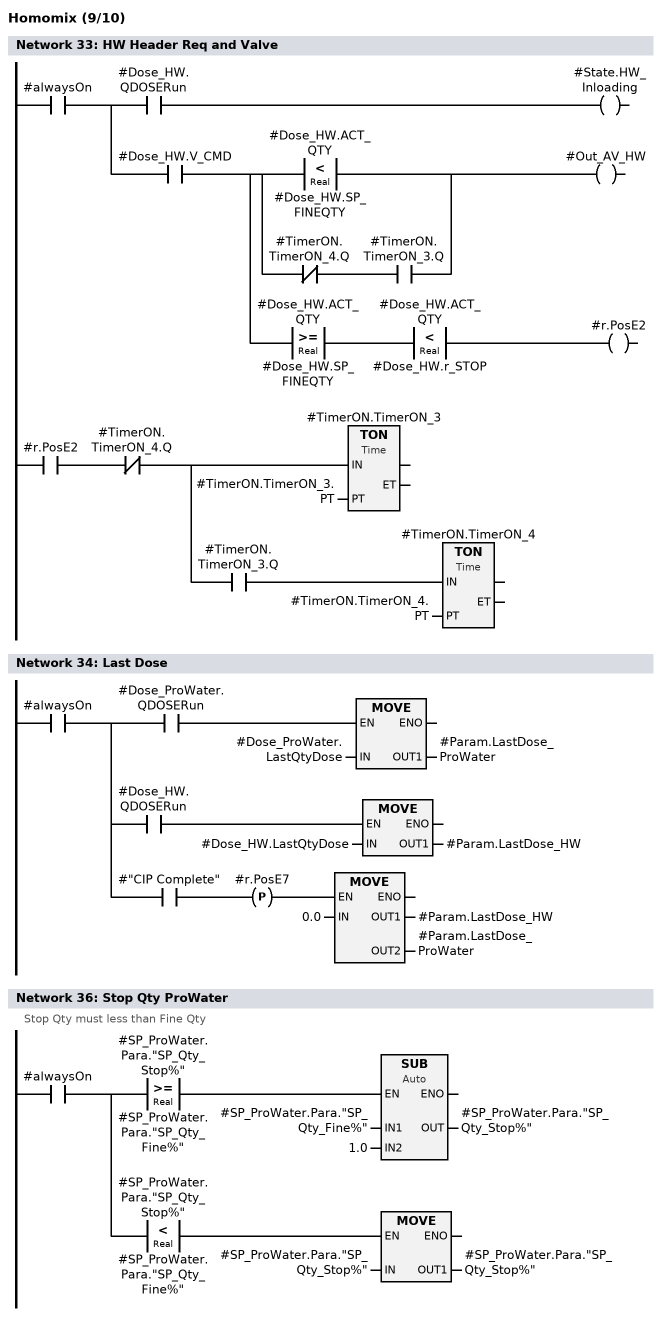
   RUNG wire#powerrail
      Contact( #alwaysOn )
      wire#w1
      Contact( #Dose_HW.QDOSERun )
      Coil( #State.HW_Inloading )
   END_RUNG
   RUNG wire#w1
      Contact( #Dose_HW.V_CMD )
      wire#w2
      { S7_Templates := "SrcType := Real" } LT_Contact(in1 := #Dose_HW.ACT_QTY, in2 := #Dose_HW.SP_FINEQTY)
      wire#w3
      Coil( #Out_AV_HW )
   END_RUNG
   RUNG wire#w2
      I_Contact( #TimerON.TimerON_4.Q )
      Contact( #TimerON.TimerON_3.Q )
   END_RUNG wire#w3
   RUNG wire#w2
      { S7_Templates := "SrcType := Real" } GE_Contact(in1 := #Dose_HW.ACT_QTY, in2 := #Dose_HW.SP_FINEQTY)
      { S7_Templates := "SrcType := Real" } LT_Contact(in1 := #Dose_HW.ACT_QTY, in2 := #Dose_HW.r_STOP)
      Coil( #r.PosE2 )
   END_RUNG
   RUNG wire#powerrail
      Contact( #r.PosE2 )
      I_Contact( #TimerON.TimerON_4.Q )
      wire#w4
      { S7_Templates := "time_type := Time" } #TimerON.TimerON_3.TON(pt := #TimerON.TimerON_3.PT, et =>)
   END_RUNG
   RUNG wire#w4
      Contact( #TimerON.TimerON_3.Q )
      { S7_Templates := "time_type := Time" } #TimerON.TimerON_4.TON(pt := #TimerON.TimerON_4.PT, et =>)
   END_RUNG
   // the same network as SCL:
   #State.HW_Inloading := #alwaysOn AND #Dose_HW.QDOSERun;
   #_w1 := #alwaysOn AND #Dose_HW.V_CMD;
   #Out_AV_HW := #_w1 AND ((#Dose_HW.ACT_QTY < #Dose_HW.SP_FINEQTY) OR (NOT #TimerON.TimerON_4.Q AND #TimerON.TimerON_3.Q));
   #r.PosE2 := #_w1 AND (#Dose_HW.ACT_QTY >= #Dose_HW.SP_FINEQTY) AND (#Dose_HW.ACT_QTY < #Dose_HW.r_STOP);
   #_w2 := #r.PosE2 AND NOT #TimerON.TimerON_4.Q;
   #TimerON.TimerON_3.TON(IN := #_w2, PT := #TimerON.TimerON_3.PT);
   #TimerON.TimerON_4.TON(IN := #_w2 AND #TimerON.TimerON_3.Q, PT := #TimerON.TimerON_4.PT);
END_REGION

REGION Network 34: Last Dose
   RUNG wire#powerrail
      Contact( #alwaysOn )
      wire#w1
      Contact( #Dose_ProWater.QDOSERun )
      Move(in := #Dose_ProWater.LastQtyDose, out1 => #Param.LastDose_ProWater)
   END_RUNG
   RUNG wire#w1
      Contact( #Dose_HW.QDOSERun )
      Move(in := #Dose_HW.LastQtyDose, out1 => #Param.LastDose_HW)
   END_RUNG
   RUNG wire#w1
      Contact( #"CIP Complete" )
      P_Trig( #r.PosE7 )
      Move(in := 0.0, out1 => #Param.LastDose_HW, out2 => #Param.LastDose_ProWater)
   END_RUNG
   // the same network as SCL:
   IF #alwaysOn AND #Dose_ProWater.QDOSERun THEN
       #Param.LastDose_ProWater := #Dose_ProWater.LastQtyDose;
   END_IF;
   IF #alwaysOn AND #Dose_HW.QDOSERun THEN #Param.LastDose_HW := #Dose_HW.LastQtyDose; END_IF;
   #_w1 := #alwaysOn AND #"CIP Complete";
   #_w2 := #_w1 AND NOT #r.PosE7;   // rising edge
   #r.PosE7 := #_w1;
   IF #_w2 THEN
       #Param.LastDose_HW := 0.0;
       #Param.LastDose_ProWater := 0.0;
   END_IF;
END_REGION

REGION Network 36: Stop Qty ProWater
   // Stop Qty must less than Fine Qty
   RUNG wire#powerrail
      Contact( #alwaysOn )
      wire#w1
      { S7_Templates := "SrcType := Real" } GE_Contact(in1 := #SP_ProWater.Para."SP_Qty_Stop%", in2 := #SP_ProWater.Para."SP_Qty_Fine%")
      Sub(in1 := #SP_ProWater.Para."SP_Qty_Fine%", in2 := 1.0, out => #SP_ProWater.Para."SP_Qty_Stop%")
   END_RUNG
   RUNG wire#w1
      { S7_Templates := "SrcType := Real" } LT_Contact(in1 := #SP_ProWater.Para."SP_Qty_Stop%", in2 := #SP_ProWater.Para."SP_Qty_Fine%")
      Move(in := #SP_ProWater.Para."SP_Qty_Stop%", out1 => #SP_ProWater.Para."SP_Qty_Stop%")
   END_RUNG
   // the same network as SCL:
   IF #alwaysOn AND (#SP_ProWater.Para."SP_Qty_Stop%" >= #SP_ProWater.Para."SP_Qty_Fine%") THEN
       #SP_ProWater.Para."SP_Qty_Stop%" := #SP_ProWater.Para."SP_Qty_Fine%" - 1.0;
   END_IF;
   IF #alwaysOn AND (#SP_ProWater.Para."SP_Qty_Stop%" < #SP_ProWater.Para."SP_Qty_Fine%") THEN
       #SP_ProWater.Para."SP_Qty_Stop%" := #SP_ProWater.Para."SP_Qty_Stop%";
   END_IF;
END_REGION

REGION Network 37: Stop Qty HW
   // Stop Qty must less than Fine Qty
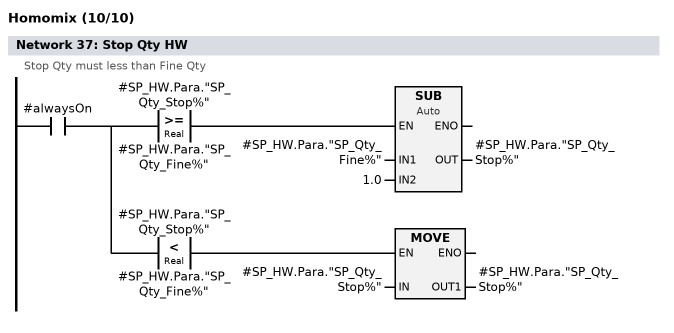
   RUNG wire#powerrail
      Contact( #alwaysOn )
      wire#w1
      { S7_Templates := "SrcType := Real" } GE_Contact(in1 := #SP_HW.Para."SP_Qty_Stop%", in2 := #SP_HW.Para."SP_Qty_Fine%")
      Sub(in1 := #SP_HW.Para."SP_Qty_Fine%", in2 := 1.0, out => #SP_HW.Para."SP_Qty_Stop%")
   END_RUNG
   RUNG wire#w1
      { S7_Templates := "SrcType := Real" } LT_Contact(in1 := #SP_HW.Para."SP_Qty_Stop%", in2 := #SP_HW.Para."SP_Qty_Fine%")
      Move(in := #SP_HW.Para."SP_Qty_Stop%", out1 => #SP_HW.Para."SP_Qty_Stop%")
   END_RUNG
   // the same network as SCL:
   IF #alwaysOn AND (#SP_HW.Para."SP_Qty_Stop%" >= #SP_HW.Para."SP_Qty_Fine%") THEN
       #SP_HW.Para."SP_Qty_Stop%" := #SP_HW.Para."SP_Qty_Fine%" - 1.0;
   END_IF;
   IF #alwaysOn AND (#SP_HW.Para."SP_Qty_Stop%" < #SP_HW.Para."SP_Qty_Fine%") THEN
       #SP_HW.Para."SP_Qty_Stop%" := #SP_HW.Para."SP_Qty_Stop%";
   END_IF;
END_REGION
END_FUNCTION_BLOCK

FUNCTION_BLOCK "Raw_Pulse"   // FB20, LAD
{ S7_Optimized_Access := 'TRUE' }
VERSION : 0.1
// stored: AutoNumber true, IsIECCheckEnabled false, IsRetainMemResEnabled false, MemoryReserve 100, SetENOAutomatically false, UDAEnableTagReadback false
   VAR_INPUT
      CountReset : Bool;
      CountMode : Bool;
      DoseRun : Bool;
      CmdStep : Int;
      FT_Pulse : Bool;   // Pulse Flow Meter
      FT_Tot : Real;
      Dose_SP : Real;
      Speed_AV : Real;
      Speed_SP : Real;
   END_VAR
   VAR_OUTPUT
      Q_FT_Star : Real;
      Q_FT_Stop : Real;
      Q_SPQty : Real;
      Q_FineQty : Real;
      Q_StopQty : Real;
      Q_P_Speed : Real;
      Q_P_FineSpeed : Real;
      Q_P_CoasSpeed : Real;
   END_VAR
   VAR_IN_OUT
      Q_FT_Tot : Real;
   END_VAR
   VAR RETAIN
      Para : Struct
         "SP_Qty_Stop%" : Real := 3.0;
         "SP_Qty_Fine%" : Real := 20.0;
         SP_Qty_Stop : Real;
         SP_Qty_Fine : Real;
         SP_Pump_Co : Real := 80.0;
         SP_Pump_Fi : Real := 20.0;
         "Pulse/Liter" : Real := 1.0;
      END_STRUCT;
   END_VAR
   VAR
      alwaysON { S7_SetPoint := 'True'} : Bool;
      DosePE : Bool;
      "BIT.FT_Pulse" : Bool;
   END_VAR
   VAR_TEMP   // added for the SCL form of the ladder/FBD networks
      _w1 : Bool;
      _w2 : Bool;
      _w3 : Bool;
      _w4 : Bool;
   END_VAR
BEGIN

REGION Network 1: alwaysON
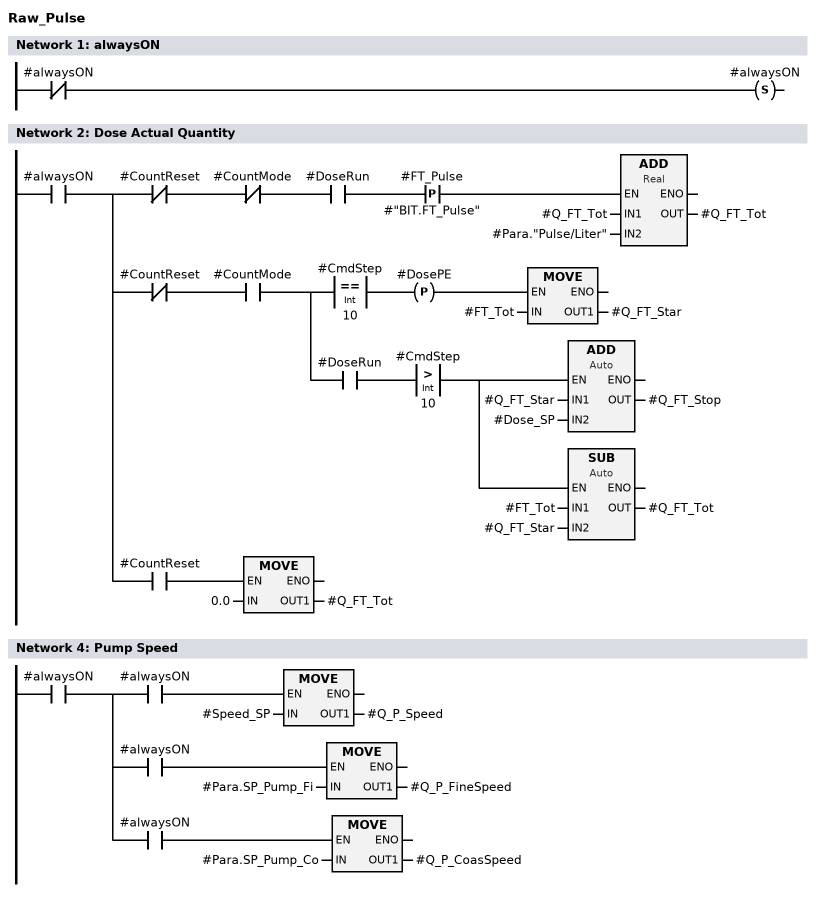
   RUNG wire#powerrail
      I_Contact( #alwaysON )
      S_Coil( #alwaysON )
   END_RUNG
   // the same network as SCL:
   IF NOT #alwaysON THEN #alwaysON := TRUE; END_IF;
END_REGION

REGION Network 2: Dose Actual Quantity
   RUNG wire#powerrail
      Contact( #alwaysON )
      wire#w1
      I_Contact( #CountReset )
      I_Contact( #CountMode )
      Contact( #DoseRun )
      P_Contact(operand := #FT_Pulse, bit := #"BIT.FT_Pulse")
      { S7_Templates := "SrcType := Real" } Add(in1 := #Q_FT_Tot, in2 := #Para."Pulse/Liter", out => #Q_FT_Tot)
   END_RUNG
   RUNG wire#w1
      I_Contact( #CountReset )
      Contact( #CountMode )
      wire#w2
      { S7_Templates := "SrcType := Int" } EQ_Contact(in1 := #CmdStep, in2 := 10)
      P_Trig( #DosePE )
      Move(in := #FT_Tot, out1 => #Q_FT_Star)
   END_RUNG
   RUNG wire#w2
      Contact( #DoseRun )
      { S7_Templates := "SrcType := Int" } GT_Contact(in1 := #CmdStep, in2 := 10)
      wire#w3
      Add(in1 := #Q_FT_Star, in2 := #Dose_SP, out => #Q_FT_Stop)
   END_RUNG
   RUNG wire#w3
      Sub(in1 := #FT_Tot, in2 := #Q_FT_Star, out => #Q_FT_Tot)
   END_RUNG
   RUNG wire#w1
      Contact( #CountReset )
      Move(in := 0.0, out1 => #Q_FT_Tot)
   END_RUNG
   // the same network as SCL:
   #_w1 := #alwaysON AND NOT #CountReset AND NOT #CountMode AND #DoseRun AND #FT_Pulse AND NOT #"BIT.FT_Pulse";   // rising edge of #FT_Pulse
   #"BIT.FT_Pulse" := #FT_Pulse;
   IF #_w1 THEN #Q_FT_Tot := #Q_FT_Tot + #Para."Pulse/Liter"; END_IF;
   #_w2 := #alwaysON AND NOT #CountReset AND #CountMode;
   #_w3 := #_w2 AND (#CmdStep = 10);
   #_w4 := #_w3 AND NOT #DosePE;   // rising edge
   #DosePE := #_w3;
   IF #_w4 THEN #Q_FT_Star := #FT_Tot; END_IF;
   IF #_w2 AND #DoseRun AND (#CmdStep > 10) THEN
       #Q_FT_Stop := #Q_FT_Star + #Dose_SP;
       #Q_FT_Tot := #FT_Tot - #Q_FT_Star;
   END_IF;
   IF #alwaysON AND #CountReset THEN #Q_FT_Tot := 0.0; END_IF;
END_REGION

NETWORK
TITLE = Quantity Calculation
// SP Quantity
      L     #Dose_SP;
      T     #Q_SPQty;
// Fine Quantity Calculation
      L     #Dose_SP;
      L     #Para."SP_Qty_Fine%";
      *R;
      L     100.0;
      /R;
      T     #Para.SP_Qty_Fine;

      L     #Dose_SP;
      L     #Para.SP_Qty_Fine;
      -R;
      T     #Q_FineQty;

// Stop Quantity Calculation
      L     #Dose_SP;
      L     #Para."SP_Qty_Stop%";
      *R;
      L     100.0;
      /R;
      T     #Para.SP_Qty_Stop;

      L     #Dose_SP;
      L     #Para.SP_Qty_Stop;
      -R;
      T     #Q_StopQty;


REGION Network 4: Pump Speed
   RUNG wire#powerrail
      Contact( #alwaysON )
      wire#w1
      Contact( #alwaysON )
      Move(in := #Speed_SP, out1 => #Q_P_Speed)
   END_RUNG
   RUNG wire#w1
      Contact( #alwaysON )
      Move(in := #Para.SP_Pump_Fi, out1 => #Q_P_FineSpeed)
   END_RUNG
   RUNG wire#w1
      Contact( #alwaysON )
      Move(in := #Para.SP_Pump_Co, out1 => #Q_P_CoasSpeed)
   END_RUNG
   // the same network as SCL:
   IF #alwaysON AND #alwaysON THEN
       #Q_P_Speed := #Speed_SP;
       #Q_P_FineSpeed := #Para.SP_Pump_Fi;
       #Q_P_CoasSpeed := #Para.SP_Pump_Co;
   END_IF;
END_REGION
END_FUNCTION_BLOCK

FUNCTION_BLOCK "IO Valve Homomixer"   // FB3, LAD
{ S7_Optimized_Access := 'FALSE' }
VERSION : 0.1
// stored: AutoNumber true, IsIECCheckEnabled false, SetENOAutomatically false, UDAEnableTagReadback false
   VAR_INPUT
      lock : Bool;
      Init : Bool;
      testing : Bool;
      Reset : Bool;
   END_VAR
   VAR
      "AV-12.01" { S7_SetPoint := 'True'} : "Valve";
      "AV-12.02" { S7_SetPoint := 'True'} : "Valve";
      "AV-12.03" { S7_SetPoint := 'True'} : "Valve";
      "AV-12.04" { S7_SetPoint := 'True'} : "Valve";
      "AV-12.05" { S7_SetPoint := 'True'} : "Valve";
      "AV-12.06" { S7_SetPoint := 'True'} : "Valve";
      "AV-12.07" { S7_SetPoint := 'True'} : "Valve";
      "AV-12.11" { S7_SetPoint := 'True'} : "Valve";
      "AV-12.12" { S7_SetPoint := 'True'} : "Valve";
      "AV-13.01" { S7_SetPoint := 'True'} : "Valve";
      "AV-13.02" { S7_SetPoint := 'True'} : "Valve";
      "AV-13.03" { S7_SetPoint := 'True'} : "Valve";
      "AV-13.04" { S7_SetPoint := 'True'} : "Valve";
      "AV-13.05" { S7_SetPoint := 'True'} : "Valve";
      "AV-13.06" { S7_SetPoint := 'True'} : "Valve";
      "AV-13.07" { S7_SetPoint := 'True'} : "Valve";
      "AV-14.01" { S7_SetPoint := 'True'} : "Valve";
      "AV-14.02" { S7_SetPoint := 'True'} : "Valve";
      "AV-14.03" { S7_SetPoint := 'True'} : "Valve";
      "AV-14.04" { S7_SetPoint := 'True'} : "Valve";
      "AV-14.05" { S7_SetPoint := 'True'} : "Valve";
      "AV-14.06" { S7_SetPoint := 'True'} : "Valve";
      "AV-14.07" { S7_SetPoint := 'True'} : "Valve";
      "P-12.01" { S7_SetPoint := 'True'} : "Motor";
      "P-13.01" { S7_SetPoint := 'True'} : "Motor";
      "P-14.01" { S7_SetPoint := 'True'} : "Motor";
   END_VAR
   // "AV-12.01".OPdwCmd := 16#0008_0000;
   // "AV-12.02".OPdwCmd := 16#0008_0000;
   // "AV-12.03".OPdwCmd := 16#0002_0000;
   // "AV-12.04".OPdwCmd := 16#0008_0000;
   // "AV-13.01".OPdwCmd := 16#0008_0000;
   // "AV-13.02".OPdwCmd := 16#0008_0000;
   // "AV-13.03".OPdwCmd := 16#0002_0000;
BEGIN

REGION Network 1 (SCL): FB OPEN and CLOSE 12
   IF #testing THEN
       // Statement section IF
       #"AV-12.01".FB_OPEN := #"AV-12.01".QCMD_OP;
       #"AV-12.01".FB_CLOSE := NOT #"AV-12.01".QCMD_OP;
       #"AV-12.02".FB_OPEN := #"AV-12.02".QCMD_OP;
       #"AV-12.02".FB_CLOSE := NOT #"AV-12.02".QCMD_OP;
       #"AV-12.03".FB_OPEN := #"AV-12.03".QCMD_OP;
       #"AV-12.03".FB_CLOSE := NOT #"AV-12.03".QCMD_OP;
       #"AV-12.04".FB_OPEN := #"AV-12.04".QCMD_OP;
       #"AV-12.04".FB_CLOSE := NOT #"AV-12.04".QCMD_OP;
       #"AV-12.05".FB_OPEN := #"AV-12.05".QCMD_OP;
       #"AV-12.05".FB_CLOSE := NOT #"AV-12.05".QCMD_OP;
       #"AV-12.06".FB_OPEN := #"AV-12.06".QCMD_OP;
       #"AV-12.06".FB_CLOSE := NOT #"AV-12.06".QCMD_OP;
       #"AV-12.07".FB_OPEN := #"AV-12.07".QCMD_OP;
       #"AV-12.07".FB_CLOSE := NOT #"AV-12.07".QCMD_OP;
       #"AV-12.11".FB_OPEN := #"AV-12.11".QCMD_OP;
       #"AV-12.11".FB_CLOSE := NOT #"AV-12.11".QCMD_OP;
       #"AV-12.12".FB_OPEN := #"AV-12.12".QCMD_OP;
       #"AV-12.12".FB_CLOSE := NOT #"AV-12.12".QCMD_OP;
   ELSE
       // Statement section ELSE
       #"AV-12.01".FB_OPEN := NOT "ZSC-12.01";
       #"AV-12.01".FB_CLOSE := "ZSC-12.01";
       #"AV-12.02".FB_OPEN := NOT "ZSC-12.02";
       #"AV-12.02".FB_CLOSE := "ZSC-12.02";
       #"AV-12.03".FB_OPEN := #"AV-12.03".QCMD_OP;
       #"AV-12.03".FB_CLOSE := NOT #"AV-12.03".QCMD_OP;
       #"AV-12.04".FB_OPEN := #"AV-12.04".QCMD_OP;
       #"AV-12.04".FB_CLOSE := NOT #"AV-12.04".QCMD_OP;
       #"AV-12.05".FB_OPEN := #"AV-12.05".QCMD_OP;
       #"AV-12.05".FB_CLOSE := NOT #"AV-12.05".QCMD_OP;
       #"AV-12.06".FB_OPEN := #"AV-12.06".QCMD_OP;
       #"AV-12.06".FB_CLOSE := NOT #"AV-12.06".QCMD_OP;
       #"AV-12.07".FB_OPEN := #"AV-12.07".QCMD_OP;
       #"AV-12.07".FB_CLOSE := NOT #"AV-12.07".QCMD_OP;
       #"AV-12.11".FB_OPEN := #"AV-12.11".QCMD_OP;
       #"AV-12.11".FB_CLOSE := NOT #"AV-12.11".QCMD_OP;
       #"AV-12.12".FB_OPEN := #"AV-12.12".QCMD_OP;
       #"AV-12.12".FB_CLOSE := NOT #"AV-12.12".QCMD_OP;
   END_IF;
END_REGION

NETWORK
TITLE = FB Monitoring Time 12
// FB OPEN Time
      L     t#20s;
      T     #"AV-12.01".MON_T;
      T     #"AV-12.02".MON_T;
      T     #"AV-12.03".MON_T;
      T     #"AV-12.04".MON_T;
      T     #"AV-12.05".MON_T;
      T     #"AV-12.06".MON_T;
      T     #"AV-12.07".MON_T;
      T     #"AV-12.11".MON_T;
      T     #"AV-12.12".MON_T;
// FB CLOSE Time
      L     t#20s;
      T     #"AV-12.01".MON_T_CLOSE;
      T     #"AV-12.02".MON_T_CLOSE;
      T     #"AV-12.03".MON_T_CLOSE;
      T     #"AV-12.04".MON_T_CLOSE;
      T     #"AV-12.05".MON_T_CLOSE;
      T     #"AV-12.06".MON_T_CLOSE;
      T     #"AV-12.07".MON_T_CLOSE;
      T     #"AV-12.11".MON_T_CLOSE;
      T     #"AV-12.12".MON_T_CLOSE;

REGION Network 3: AV-12.01 w ZSC
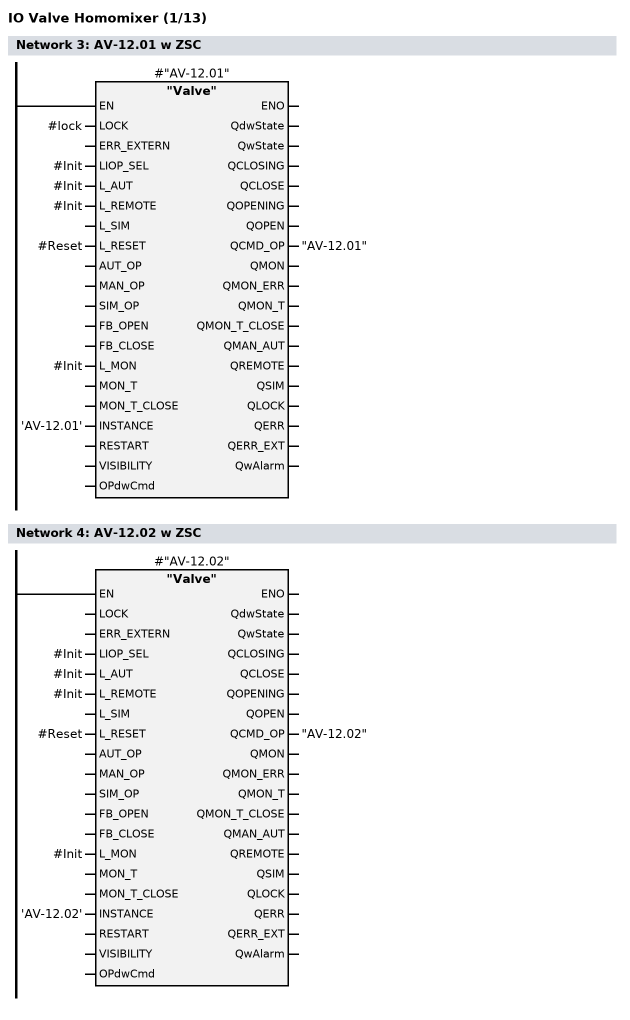
   RUNG wire#powerrail
      #"AV-12.01"(LOCK := #lock, ERR_EXTERN :=, LIOP_SEL := #Init, L_AUT := #Init, L_REMOTE := #Init, L_SIM :=, L_RESET := #Reset, AUT_OP :=, MAN_OP :=, SIM_OP :=, FB_OPEN :=, FB_CLOSE :=, L_MON := #Init, MON_T :=, MON_T_CLOSE :=, INSTANCE := 'AV-12.01', RESTART :=, VISIBILITY :=, OPdwCmd :=, QdwState =>, QwState =>, QCLOSING =>, QCLOSE =>, QOPENING =>, QOPEN =>, QCMD_OP => "AV-12.01", QMON =>, QMON_ERR =>, QMON_T =>, QMON_T_CLOSE =>, QMAN_AUT =>, QREMOTE =>, QSIM =>, QLOCK =>, QERR =>, QERR_EXT =>, QwAlarm =>)
   END_RUNG
   // the same network as SCL:
   #"AV-12.01"(LOCK := #lock,   // "Valve"
               LIOP_SEL := #Init,
               L_AUT := #Init,
               L_REMOTE := #Init,
               L_RESET := #Reset,
               L_MON := #Init,
               INSTANCE := 'AV-12.01',
               QCMD_OP => "AV-12.01");
END_REGION

REGION Network 4: AV-12.02 w ZSC
   RUNG wire#powerrail
      #"AV-12.02"(LOCK :=, ERR_EXTERN :=, LIOP_SEL := #Init, L_AUT := #Init, L_REMOTE := #Init, L_SIM :=, L_RESET := #Reset, AUT_OP :=, MAN_OP :=, SIM_OP :=, FB_OPEN :=, FB_CLOSE :=, L_MON := #Init, MON_T :=, MON_T_CLOSE :=, INSTANCE := 'AV-12.02', RESTART :=, VISIBILITY :=, OPdwCmd :=, QdwState =>, QwState =>, QCLOSING =>, QCLOSE =>, QOPENING =>, QOPEN =>, QCMD_OP => "AV-12.02", QMON =>, QMON_ERR =>, QMON_T =>, QMON_T_CLOSE =>, QMAN_AUT =>, QREMOTE =>, QSIM =>, QLOCK =>, QERR =>, QERR_EXT =>, QwAlarm =>)
   END_RUNG
   // the same network as SCL:
   #"AV-12.02"(LIOP_SEL := #Init,   // "Valve"
               L_AUT := #Init,
               L_REMOTE := #Init,
               L_RESET := #Reset,
               L_MON := #Init,
               INSTANCE := 'AV-12.02',
               QCMD_OP => "AV-12.02");
END_REGION

REGION Network 5: AV-12.03
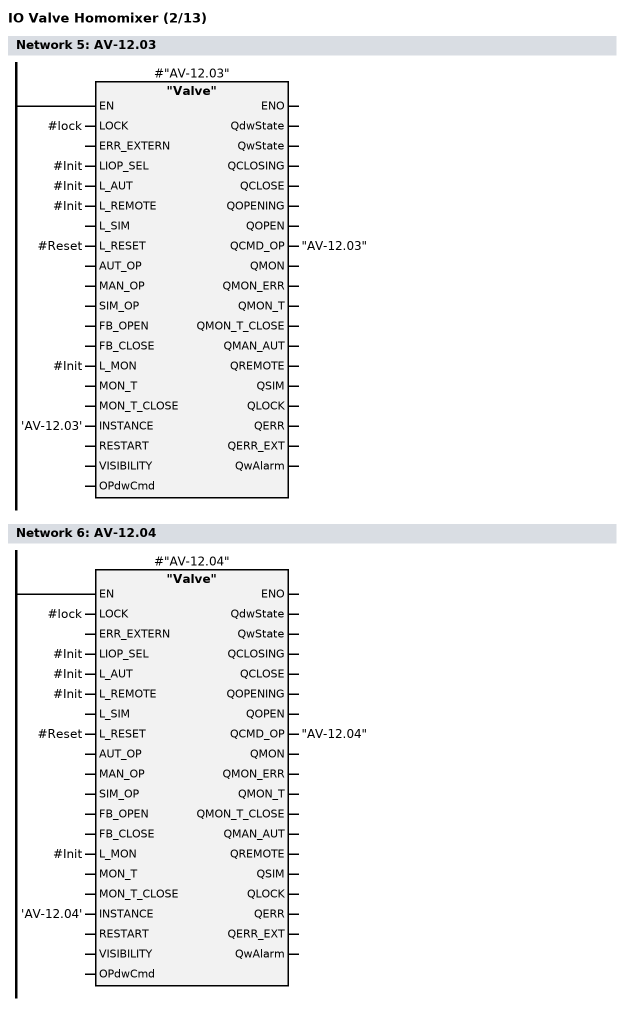
   RUNG wire#powerrail
      #"AV-12.03"(LOCK := #lock, ERR_EXTERN :=, LIOP_SEL := #Init, L_AUT := #Init, L_REMOTE := #Init, L_SIM :=, L_RESET := #Reset, AUT_OP :=, MAN_OP :=, SIM_OP :=, FB_OPEN :=, FB_CLOSE :=, L_MON := #Init, MON_T :=, MON_T_CLOSE :=, INSTANCE := 'AV-12.03', RESTART :=, VISIBILITY :=, OPdwCmd :=, QdwState =>, QwState =>, QCLOSING =>, QCLOSE =>, QOPENING =>, QOPEN =>, QCMD_OP => "AV-12.03", QMON =>, QMON_ERR =>, QMON_T =>, QMON_T_CLOSE =>, QMAN_AUT =>, QREMOTE =>, QSIM =>, QLOCK =>, QERR =>, QERR_EXT =>, QwAlarm =>)
   END_RUNG
   // the same network as SCL:
   #"AV-12.03"(LOCK := #lock,   // "Valve"
               LIOP_SEL := #Init,
               L_AUT := #Init,
               L_REMOTE := #Init,
               L_RESET := #Reset,
               L_MON := #Init,
               INSTANCE := 'AV-12.03',
               QCMD_OP => "AV-12.03");
END_REGION

REGION Network 6: AV-12.04
   RUNG wire#powerrail
      #"AV-12.04"(LOCK := #lock, ERR_EXTERN :=, LIOP_SEL := #Init, L_AUT := #Init, L_REMOTE := #Init, L_SIM :=, L_RESET := #Reset, AUT_OP :=, MAN_OP :=, SIM_OP :=, FB_OPEN :=, FB_CLOSE :=, L_MON := #Init, MON_T :=, MON_T_CLOSE :=, INSTANCE := 'AV-12.04', RESTART :=, VISIBILITY :=, OPdwCmd :=, QdwState =>, QwState =>, QCLOSING =>, QCLOSE =>, QOPENING =>, QOPEN =>, QCMD_OP => "AV-12.04", QMON =>, QMON_ERR =>, QMON_T =>, QMON_T_CLOSE =>, QMAN_AUT =>, QREMOTE =>, QSIM =>, QLOCK =>, QERR =>, QERR_EXT =>, QwAlarm =>)
   END_RUNG
   // the same network as SCL:
   #"AV-12.04"(LOCK := #lock,   // "Valve"
               LIOP_SEL := #Init,
               L_AUT := #Init,
               L_REMOTE := #Init,
               L_RESET := #Reset,
               L_MON := #Init,
               INSTANCE := 'AV-12.04',
               QCMD_OP => "AV-12.04");
END_REGION

REGION Network 7: AV-12.05
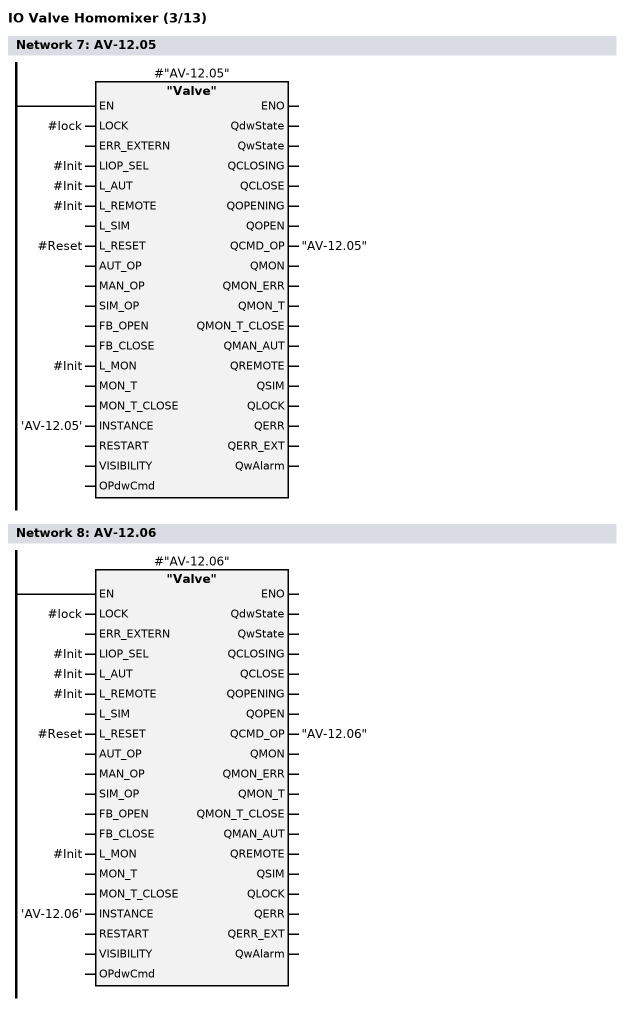
   RUNG wire#powerrail
      #"AV-12.05"(LOCK := #lock, ERR_EXTERN :=, LIOP_SEL := #Init, L_AUT := #Init, L_REMOTE := #Init, L_SIM :=, L_RESET := #Reset, AUT_OP :=, MAN_OP :=, SIM_OP :=, FB_OPEN :=, FB_CLOSE :=, L_MON := #Init, MON_T :=, MON_T_CLOSE :=, INSTANCE := 'AV-12.05', RESTART :=, VISIBILITY :=, OPdwCmd :=, QdwState =>, QwState =>, QCLOSING =>, QCLOSE =>, QOPENING =>, QOPEN =>, QCMD_OP => "AV-12.05", QMON =>, QMON_ERR =>, QMON_T =>, QMON_T_CLOSE =>, QMAN_AUT =>, QREMOTE =>, QSIM =>, QLOCK =>, QERR =>, QERR_EXT =>, QwAlarm =>)
   END_RUNG
   // the same network as SCL:
   #"AV-12.05"(LOCK := #lock,   // "Valve"
               LIOP_SEL := #Init,
               L_AUT := #Init,
               L_REMOTE := #Init,
               L_RESET := #Reset,
               L_MON := #Init,
               INSTANCE := 'AV-12.05',
               QCMD_OP => "AV-12.05");
END_REGION

REGION Network 8: AV-12.06
   RUNG wire#powerrail
      #"AV-12.06"(LOCK := #lock, ERR_EXTERN :=, LIOP_SEL := #Init, L_AUT := #Init, L_REMOTE := #Init, L_SIM :=, L_RESET := #Reset, AUT_OP :=, MAN_OP :=, SIM_OP :=, FB_OPEN :=, FB_CLOSE :=, L_MON := #Init, MON_T :=, MON_T_CLOSE :=, INSTANCE := 'AV-12.06', RESTART :=, VISIBILITY :=, OPdwCmd :=, QdwState =>, QwState =>, QCLOSING =>, QCLOSE =>, QOPENING =>, QOPEN =>, QCMD_OP => "AV-12.06", QMON =>, QMON_ERR =>, QMON_T =>, QMON_T_CLOSE =>, QMAN_AUT =>, QREMOTE =>, QSIM =>, QLOCK =>, QERR =>, QERR_EXT =>, QwAlarm =>)
   END_RUNG
   // the same network as SCL:
   #"AV-12.06"(LOCK := #lock,   // "Valve"
               LIOP_SEL := #Init,
               L_AUT := #Init,
               L_REMOTE := #Init,
               L_RESET := #Reset,
               L_MON := #Init,
               INSTANCE := 'AV-12.06',
               QCMD_OP => "AV-12.06");
END_REGION

REGION Network 9: AV-12.07
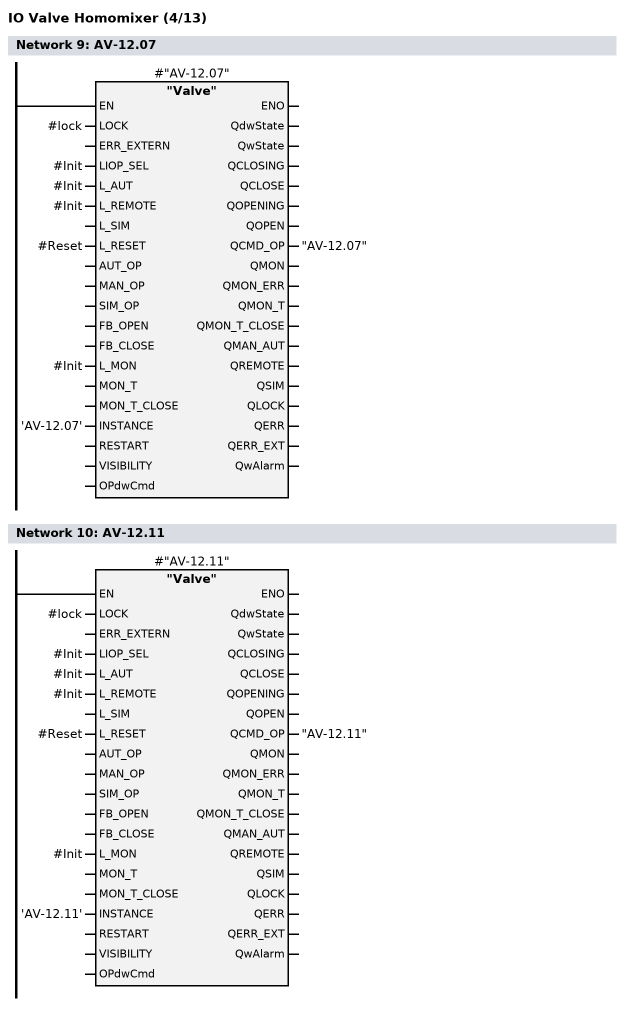
   RUNG wire#powerrail
      #"AV-12.07"(LOCK := #lock, ERR_EXTERN :=, LIOP_SEL := #Init, L_AUT := #Init, L_REMOTE := #Init, L_SIM :=, L_RESET := #Reset, AUT_OP :=, MAN_OP :=, SIM_OP :=, FB_OPEN :=, FB_CLOSE :=, L_MON := #Init, MON_T :=, MON_T_CLOSE :=, INSTANCE := 'AV-12.07', RESTART :=, VISIBILITY :=, OPdwCmd :=, QdwState =>, QwState =>, QCLOSING =>, QCLOSE =>, QOPENING =>, QOPEN =>, QCMD_OP => "AV-12.07", QMON =>, QMON_ERR =>, QMON_T =>, QMON_T_CLOSE =>, QMAN_AUT =>, QREMOTE =>, QSIM =>, QLOCK =>, QERR =>, QERR_EXT =>, QwAlarm =>)
   END_RUNG
   // the same network as SCL:
   #"AV-12.07"(LOCK := #lock,   // "Valve"
               LIOP_SEL := #Init,
               L_AUT := #Init,
               L_REMOTE := #Init,
               L_RESET := #Reset,
               L_MON := #Init,
               INSTANCE := 'AV-12.07',
               QCMD_OP => "AV-12.07");
END_REGION

REGION Network 10: AV-12.11
   RUNG wire#powerrail
      #"AV-12.11"(LOCK := #lock, ERR_EXTERN :=, LIOP_SEL := #Init, L_AUT := #Init, L_REMOTE := #Init, L_SIM :=, L_RESET := #Reset, AUT_OP :=, MAN_OP :=, SIM_OP :=, FB_OPEN :=, FB_CLOSE :=, L_MON := #Init, MON_T :=, MON_T_CLOSE :=, INSTANCE := 'AV-12.11', RESTART :=, VISIBILITY :=, OPdwCmd :=, QdwState =>, QwState =>, QCLOSING =>, QCLOSE =>, QOPENING =>, QOPEN =>, QCMD_OP => "AV-12.11", QMON =>, QMON_ERR =>, QMON_T =>, QMON_T_CLOSE =>, QMAN_AUT =>, QREMOTE =>, QSIM =>, QLOCK =>, QERR =>, QERR_EXT =>, QwAlarm =>)
   END_RUNG
   // the same network as SCL:
   #"AV-12.11"(LOCK := #lock,   // "Valve"
               LIOP_SEL := #Init,
               L_AUT := #Init,
               L_REMOTE := #Init,
               L_RESET := #Reset,
               L_MON := #Init,
               INSTANCE := 'AV-12.11',
               QCMD_OP => "AV-12.11");
END_REGION

REGION Network 11: AV-12.12
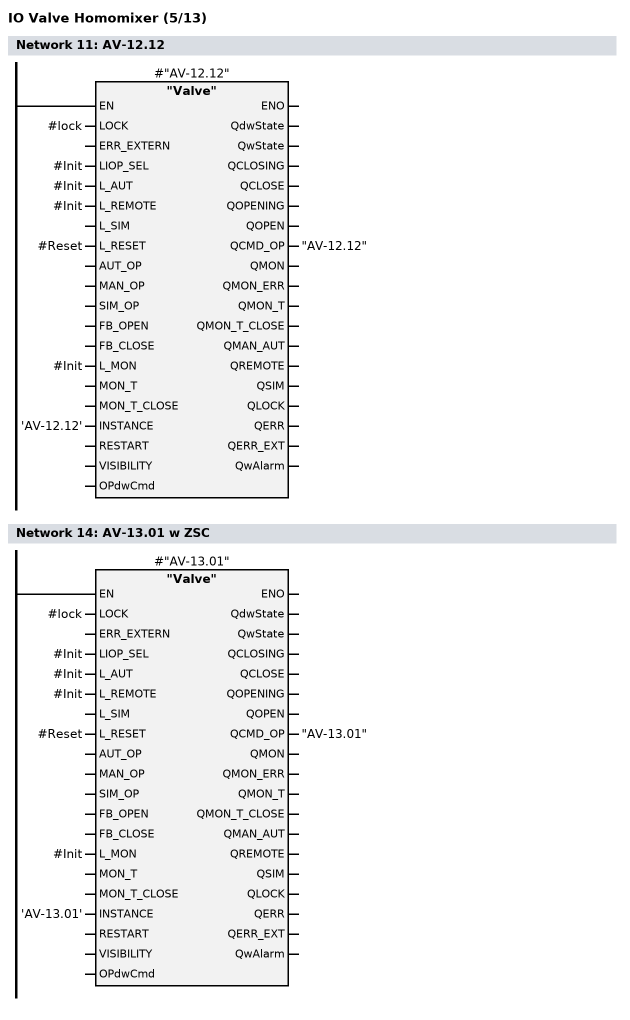
   RUNG wire#powerrail
      #"AV-12.12"(LOCK := #lock, ERR_EXTERN :=, LIOP_SEL := #Init, L_AUT := #Init, L_REMOTE := #Init, L_SIM :=, L_RESET := #Reset, AUT_OP :=, MAN_OP :=, SIM_OP :=, FB_OPEN :=, FB_CLOSE :=, L_MON := #Init, MON_T :=, MON_T_CLOSE :=, INSTANCE := 'AV-12.12', RESTART :=, VISIBILITY :=, OPdwCmd :=, QdwState =>, QwState =>, QCLOSING =>, QCLOSE =>, QOPENING =>, QOPEN =>, QCMD_OP => "AV-12.12", QMON =>, QMON_ERR =>, QMON_T =>, QMON_T_CLOSE =>, QMAN_AUT =>, QREMOTE =>, QSIM =>, QLOCK =>, QERR =>, QERR_EXT =>, QwAlarm =>)
   END_RUNG
   // the same network as SCL:
   #"AV-12.12"(LOCK := #lock,   // "Valve"
               LIOP_SEL := #Init,
               L_AUT := #Init,
               L_REMOTE := #Init,
               L_RESET := #Reset,
               L_MON := #Init,
               INSTANCE := 'AV-12.12',
               QCMD_OP => "AV-12.12");
END_REGION

REGION Network 12 (SCL): FB OPEN and CLOSE 13
   IF #testing THEN
       // Statement section IF
       #"AV-13.01".FB_OPEN := #"AV-13.01".QCMD_OP;
       #"AV-13.01".FB_CLOSE := NOT #"AV-13.01".QCMD_OP;
       #"AV-13.02".FB_OPEN := #"AV-13.02".QCMD_OP;
       #"AV-13.02".FB_CLOSE := NOT #"AV-13.02".QCMD_OP;
       #"AV-13.03".FB_OPEN := #"AV-13.03".QCMD_OP;
       #"AV-13.03".FB_CLOSE := NOT #"AV-13.03".QCMD_OP;
       #"AV-13.04".FB_OPEN := #"AV-13.04".QCMD_OP;
       #"AV-13.04".FB_CLOSE := NOT #"AV-13.04".QCMD_OP;
       #"AV-13.05".FB_OPEN := #"AV-13.05".QCMD_OP;
       #"AV-13.05".FB_CLOSE := NOT #"AV-13.05".QCMD_OP;
       #"AV-13.06".FB_OPEN := #"AV-13.06".QCMD_OP;
       #"AV-13.06".FB_CLOSE := NOT #"AV-13.06".QCMD_OP;
       #"AV-13.07".FB_OPEN := #"AV-13.07".QCMD_OP;
       #"AV-13.07".FB_CLOSE := NOT #"AV-13.07".QCMD_OP;
   ELSE
       // Statement section ELSE
       #"AV-13.01".FB_OPEN := NOT "ZSC-13.01";
       #"AV-13.01".FB_CLOSE := "ZSC-13.01";
       #"AV-13.02".FB_OPEN := NOT "ZSC-13.02";
       #"AV-13.02".FB_CLOSE := "ZSC-13.02";
       #"AV-13.03".FB_OPEN := #"AV-13.03".QCMD_OP;
       #"AV-13.03".FB_CLOSE := NOT #"AV-13.03".QCMD_OP;
       #"AV-13.04".FB_OPEN := #"AV-13.04".QCMD_OP;
       #"AV-13.04".FB_CLOSE := NOT #"AV-13.04".QCMD_OP;
       #"AV-13.05".FB_OPEN := #"AV-13.05".QCMD_OP;
       #"AV-13.05".FB_CLOSE := NOT #"AV-13.05".QCMD_OP;
       #"AV-13.06".FB_OPEN := #"AV-13.06".QCMD_OP;
       #"AV-13.06".FB_CLOSE := NOT #"AV-13.06".QCMD_OP;
       #"AV-13.07".FB_OPEN := #"AV-13.07".QCMD_OP;
       #"AV-13.07".FB_CLOSE := NOT #"AV-13.07".QCMD_OP;
   END_IF;
END_REGION

NETWORK
TITLE = FB Monitoring Time 13
// FB OPEN Time
      L     t#20s;
      T     #"AV-13.01".MON_T;
      T     #"AV-13.02".MON_T;
      T     #"AV-13.03".MON_T;
      T     #"AV-13.04".MON_T;
      T     #"AV-13.05".MON_T;
      T     #"AV-13.06".MON_T;
      T     #"AV-13.07".MON_T;
// FB CLOSE Time
      L     t#20s;
      T     #"AV-13.01".MON_T_CLOSE;
      T     #"AV-13.02".MON_T_CLOSE;
      T     #"AV-13.03".MON_T_CLOSE;
      T     #"AV-13.04".MON_T_CLOSE;
      T     #"AV-13.05".MON_T_CLOSE;
      T     #"AV-13.06".MON_T_CLOSE;
      T     #"AV-13.07".MON_T_CLOSE;

REGION Network 14: AV-13.01 w ZSC
   RUNG wire#powerrail
      #"AV-13.01"(LOCK := #lock, ERR_EXTERN :=, LIOP_SEL := #Init, L_AUT := #Init, L_REMOTE := #Init, L_SIM :=, L_RESET := #Reset, AUT_OP :=, MAN_OP :=, SIM_OP :=, FB_OPEN :=, FB_CLOSE :=, L_MON := #Init, MON_T :=, MON_T_CLOSE :=, INSTANCE := 'AV-13.01', RESTART :=, VISIBILITY :=, OPdwCmd :=, QdwState =>, QwState =>, QCLOSING =>, QCLOSE =>, QOPENING =>, QOPEN =>, QCMD_OP => "AV-13.01", QMON =>, QMON_ERR =>, QMON_T =>, QMON_T_CLOSE =>, QMAN_AUT =>, QREMOTE =>, QSIM =>, QLOCK =>, QERR =>, QERR_EXT =>, QwAlarm =>)
   END_RUNG
   // the same network as SCL:
   #"AV-13.01"(LOCK := #lock,   // "Valve"
               LIOP_SEL := #Init,
               L_AUT := #Init,
               L_REMOTE := #Init,
               L_RESET := #Reset,
               L_MON := #Init,
               INSTANCE := 'AV-13.01',
               QCMD_OP => "AV-13.01");
END_REGION

REGION Network 15: AV-13.02 w ZSC
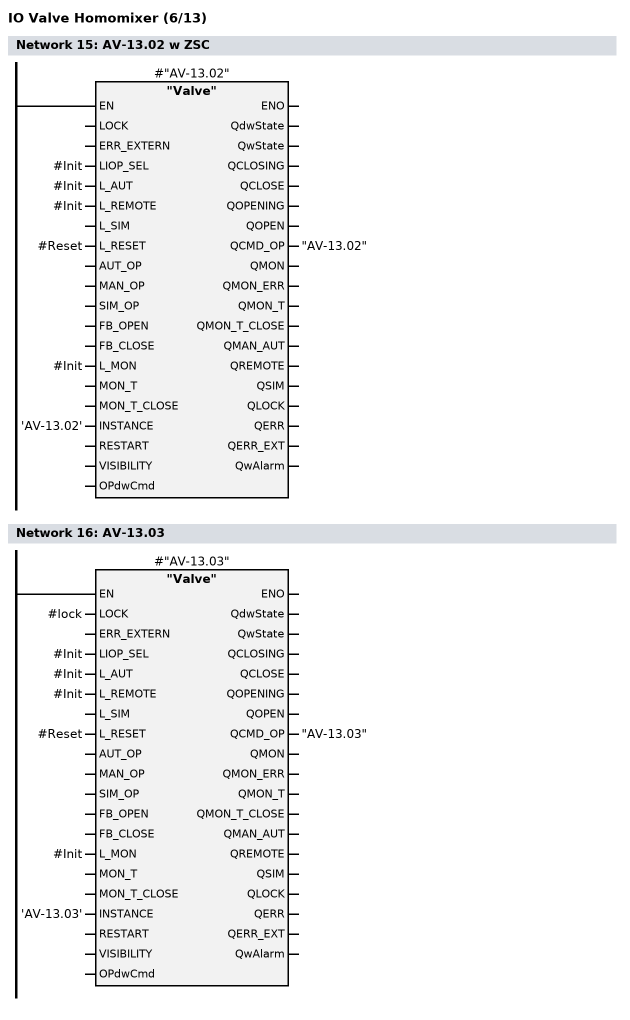
   RUNG wire#powerrail
      #"AV-13.02"(LOCK :=, ERR_EXTERN :=, LIOP_SEL := #Init, L_AUT := #Init, L_REMOTE := #Init, L_SIM :=, L_RESET := #Reset, AUT_OP :=, MAN_OP :=, SIM_OP :=, FB_OPEN :=, FB_CLOSE :=, L_MON := #Init, MON_T :=, MON_T_CLOSE :=, INSTANCE := 'AV-13.02', RESTART :=, VISIBILITY :=, OPdwCmd :=, QdwState =>, QwState =>, QCLOSING =>, QCLOSE =>, QOPENING =>, QOPEN =>, QCMD_OP => "AV-13.02", QMON =>, QMON_ERR =>, QMON_T =>, QMON_T_CLOSE =>, QMAN_AUT =>, QREMOTE =>, QSIM =>, QLOCK =>, QERR =>, QERR_EXT =>, QwAlarm =>)
   END_RUNG
   // the same network as SCL:
   #"AV-13.02"(LIOP_SEL := #Init,   // "Valve"
               L_AUT := #Init,
               L_REMOTE := #Init,
               L_RESET := #Reset,
               L_MON := #Init,
               INSTANCE := 'AV-13.02',
               QCMD_OP => "AV-13.02");
END_REGION

REGION Network 16: AV-13.03
   RUNG wire#powerrail
      #"AV-13.03"(LOCK := #lock, ERR_EXTERN :=, LIOP_SEL := #Init, L_AUT := #Init, L_REMOTE := #Init, L_SIM :=, L_RESET := #Reset, AUT_OP :=, MAN_OP :=, SIM_OP :=, FB_OPEN :=, FB_CLOSE :=, L_MON := #Init, MON_T :=, MON_T_CLOSE :=, INSTANCE := 'AV-13.03', RESTART :=, VISIBILITY :=, OPdwCmd :=, QdwState =>, QwState =>, QCLOSING =>, QCLOSE =>, QOPENING =>, QOPEN =>, QCMD_OP => "AV-13.03", QMON =>, QMON_ERR =>, QMON_T =>, QMON_T_CLOSE =>, QMAN_AUT =>, QREMOTE =>, QSIM =>, QLOCK =>, QERR =>, QERR_EXT =>, QwAlarm =>)
   END_RUNG
   // the same network as SCL:
   #"AV-13.03"(LOCK := #lock,   // "Valve"
               LIOP_SEL := #Init,
               L_AUT := #Init,
               L_REMOTE := #Init,
               L_RESET := #Reset,
               L_MON := #Init,
               INSTANCE := 'AV-13.03',
               QCMD_OP => "AV-13.03");
END_REGION

REGION Network 17: AV-13.04
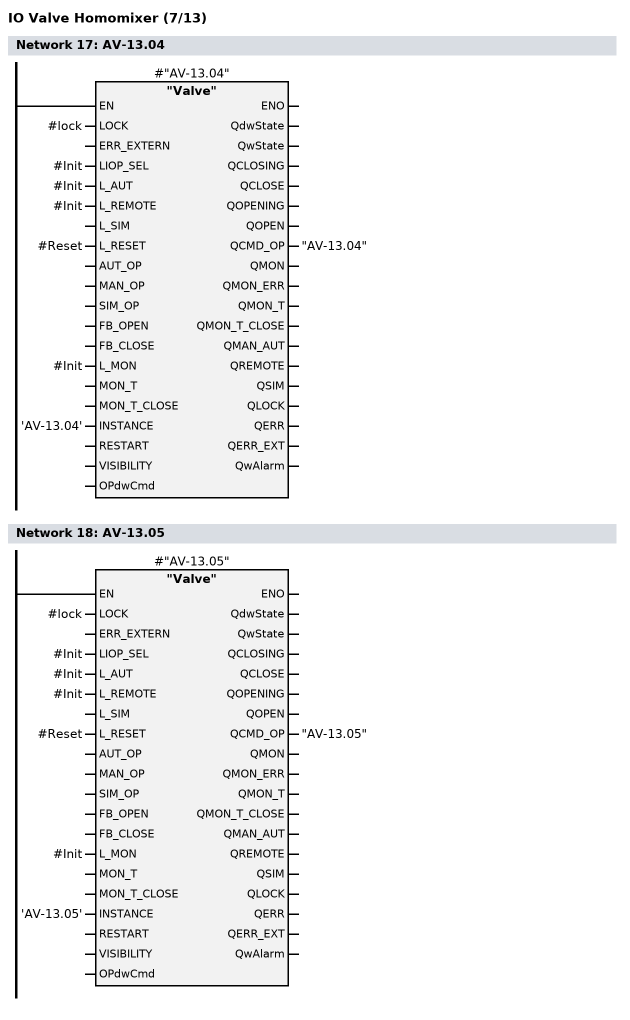
   RUNG wire#powerrail
      #"AV-13.04"(LOCK := #lock, ERR_EXTERN :=, LIOP_SEL := #Init, L_AUT := #Init, L_REMOTE := #Init, L_SIM :=, L_RESET := #Reset, AUT_OP :=, MAN_OP :=, SIM_OP :=, FB_OPEN :=, FB_CLOSE :=, L_MON := #Init, MON_T :=, MON_T_CLOSE :=, INSTANCE := 'AV-13.04', RESTART :=, VISIBILITY :=, OPdwCmd :=, QdwState =>, QwState =>, QCLOSING =>, QCLOSE =>, QOPENING =>, QOPEN =>, QCMD_OP => "AV-13.04", QMON =>, QMON_ERR =>, QMON_T =>, QMON_T_CLOSE =>, QMAN_AUT =>, QREMOTE =>, QSIM =>, QLOCK =>, QERR =>, QERR_EXT =>, QwAlarm =>)
   END_RUNG
   // the same network as SCL:
   #"AV-13.04"(LOCK := #lock,   // "Valve"
               LIOP_SEL := #Init,
               L_AUT := #Init,
               L_REMOTE := #Init,
               L_RESET := #Reset,
               L_MON := #Init,
               INSTANCE := 'AV-13.04',
               QCMD_OP => "AV-13.04");
END_REGION

REGION Network 18: AV-13.05
   RUNG wire#powerrail
      #"AV-13.05"(LOCK := #lock, ERR_EXTERN :=, LIOP_SEL := #Init, L_AUT := #Init, L_REMOTE := #Init, L_SIM :=, L_RESET := #Reset, AUT_OP :=, MAN_OP :=, SIM_OP :=, FB_OPEN :=, FB_CLOSE :=, L_MON := #Init, MON_T :=, MON_T_CLOSE :=, INSTANCE := 'AV-13.05', RESTART :=, VISIBILITY :=, OPdwCmd :=, QdwState =>, QwState =>, QCLOSING =>, QCLOSE =>, QOPENING =>, QOPEN =>, QCMD_OP => "AV-13.05", QMON =>, QMON_ERR =>, QMON_T =>, QMON_T_CLOSE =>, QMAN_AUT =>, QREMOTE =>, QSIM =>, QLOCK =>, QERR =>, QERR_EXT =>, QwAlarm =>)
   END_RUNG
   // the same network as SCL:
   #"AV-13.05"(LOCK := #lock,   // "Valve"
               LIOP_SEL := #Init,
               L_AUT := #Init,
               L_REMOTE := #Init,
               L_RESET := #Reset,
               L_MON := #Init,
               INSTANCE := 'AV-13.05',
               QCMD_OP => "AV-13.05");
END_REGION

REGION Network 19: AV-13.06
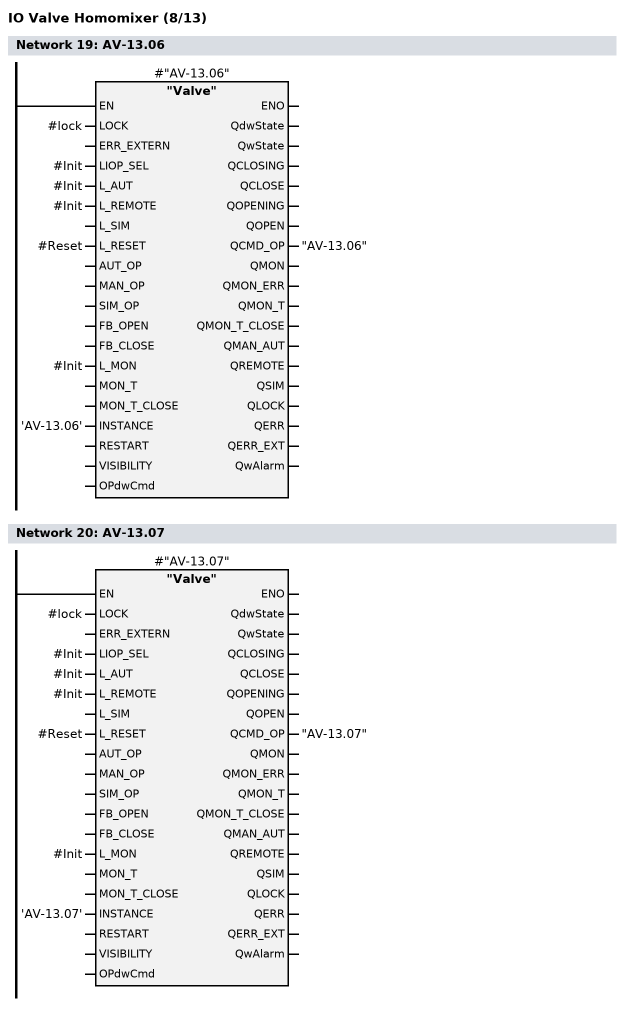
   RUNG wire#powerrail
      #"AV-13.06"(LOCK := #lock, ERR_EXTERN :=, LIOP_SEL := #Init, L_AUT := #Init, L_REMOTE := #Init, L_SIM :=, L_RESET := #Reset, AUT_OP :=, MAN_OP :=, SIM_OP :=, FB_OPEN :=, FB_CLOSE :=, L_MON := #Init, MON_T :=, MON_T_CLOSE :=, INSTANCE := 'AV-13.06', RESTART :=, VISIBILITY :=, OPdwCmd :=, QdwState =>, QwState =>, QCLOSING =>, QCLOSE =>, QOPENING =>, QOPEN =>, QCMD_OP => "AV-13.06", QMON =>, QMON_ERR =>, QMON_T =>, QMON_T_CLOSE =>, QMAN_AUT =>, QREMOTE =>, QSIM =>, QLOCK =>, QERR =>, QERR_EXT =>, QwAlarm =>)
   END_RUNG
   // the same network as SCL:
   #"AV-13.06"(LOCK := #lock,   // "Valve"
               LIOP_SEL := #Init,
               L_AUT := #Init,
               L_REMOTE := #Init,
               L_RESET := #Reset,
               L_MON := #Init,
               INSTANCE := 'AV-13.06',
               QCMD_OP => "AV-13.06");
END_REGION

REGION Network 20: AV-13.07
   RUNG wire#powerrail
      #"AV-13.07"(LOCK := #lock, ERR_EXTERN :=, LIOP_SEL := #Init, L_AUT := #Init, L_REMOTE := #Init, L_SIM :=, L_RESET := #Reset, AUT_OP :=, MAN_OP :=, SIM_OP :=, FB_OPEN :=, FB_CLOSE :=, L_MON := #Init, MON_T :=, MON_T_CLOSE :=, INSTANCE := 'AV-13.07', RESTART :=, VISIBILITY :=, OPdwCmd :=, QdwState =>, QwState =>, QCLOSING =>, QCLOSE =>, QOPENING =>, QOPEN =>, QCMD_OP => "AV-13.07", QMON =>, QMON_ERR =>, QMON_T =>, QMON_T_CLOSE =>, QMAN_AUT =>, QREMOTE =>, QSIM =>, QLOCK =>, QERR =>, QERR_EXT =>, QwAlarm =>)
   END_RUNG
   // the same network as SCL:
   #"AV-13.07"(LOCK := #lock,   // "Valve"
               LIOP_SEL := #Init,
               L_AUT := #Init,
               L_REMOTE := #Init,
               L_RESET := #Reset,
               L_MON := #Init,
               INSTANCE := 'AV-13.07',
               QCMD_OP => "AV-13.07");
END_REGION

REGION Network 21 (SCL): FB OPEN and CLOSE 14
   IF #testing THEN
       // Statement section IF
       #"AV-14.01".FB_OPEN := #"AV-14.01".QCMD_OP;
       #"AV-14.01".FB_CLOSE := NOT #"AV-14.01".QCMD_OP;
       #"AV-14.02".FB_OPEN := #"AV-14.02".QCMD_OP;
       #"AV-14.02".FB_CLOSE := NOT #"AV-14.02".QCMD_OP;
       #"AV-14.03".FB_OPEN := #"AV-14.03".QCMD_OP;
       #"AV-14.03".FB_CLOSE := NOT #"AV-14.03".QCMD_OP;
       #"AV-14.04".FB_OPEN := #"AV-14.04".QCMD_OP;
       #"AV-14.04".FB_CLOSE := NOT #"AV-14.04".QCMD_OP;
       #"AV-14.05".FB_OPEN := #"AV-14.05".QCMD_OP;
       #"AV-14.05".FB_CLOSE := NOT #"AV-14.05".QCMD_OP;
       #"AV-14.06".FB_OPEN := #"AV-14.06".QCMD_OP;
       #"AV-14.06".FB_CLOSE := NOT #"AV-14.06".QCMD_OP;
       #"AV-14.07".FB_OPEN := #"AV-14.07".QCMD_OP;
       #"AV-14.07".FB_CLOSE := NOT #"AV-14.07".QCMD_OP;
   ELSE
       // Statement section ELSE
       #"AV-14.01".FB_OPEN := NOT "ZSC-14.01";
       #"AV-14.01".FB_CLOSE := "ZSC-14.01";
       #"AV-14.02".FB_OPEN := NOT "ZSC-14.02";
       #"AV-14.02".FB_CLOSE := "ZSC-14.02";
       #"AV-14.03".FB_OPEN := #"AV-14.03".QCMD_OP;
       #"AV-14.03".FB_CLOSE := NOT #"AV-14.03".QCMD_OP;
       #"AV-14.04".FB_OPEN := #"AV-14.04".QCMD_OP;
       #"AV-14.04".FB_CLOSE := NOT #"AV-14.04".QCMD_OP;
       #"AV-14.05".FB_OPEN := #"AV-14.05".QCMD_OP;
       #"AV-14.05".FB_CLOSE := NOT #"AV-14.05".QCMD_OP;
       #"AV-14.06".FB_OPEN := #"AV-14.06".QCMD_OP;
       #"AV-14.06".FB_CLOSE := NOT #"AV-14.06".QCMD_OP;
       #"AV-14.07".FB_OPEN := #"AV-14.07".QCMD_OP;
       #"AV-14.07".FB_CLOSE := NOT #"AV-14.07".QCMD_OP;
   END_IF;
END_REGION

NETWORK
TITLE = FB Monitoring Time 14
// FB OPEN Time
      L     t#20s;
      T     #"AV-14.01".MON_T;
      T     #"AV-14.02".MON_T;
      T     #"AV-14.03".MON_T;
      T     #"AV-14.04".MON_T;
      T     #"AV-14.05".MON_T;
      T     #"AV-14.06".MON_T;
      T     #"AV-14.07".MON_T;
// FB CLOSE Time
      L     t#20s;
      T     #"AV-14.01".MON_T_CLOSE;
      T     #"AV-14.02".MON_T_CLOSE;
      T     #"AV-14.03".MON_T_CLOSE;
      T     #"AV-14.04".MON_T_CLOSE;
      T     #"AV-14.05".MON_T_CLOSE;
      T     #"AV-14.06".MON_T_CLOSE;
      T     #"AV-14.07".MON_T_CLOSE;

REGION Network 23: AV-14.01 w ZSC
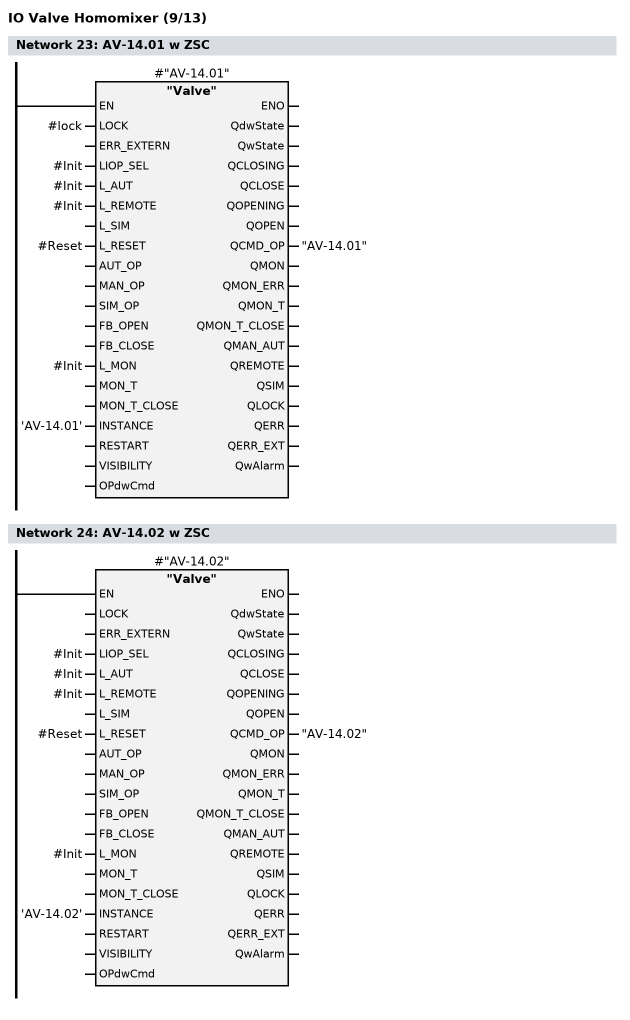
   RUNG wire#powerrail
      #"AV-14.01"(LOCK := #lock, ERR_EXTERN :=, LIOP_SEL := #Init, L_AUT := #Init, L_REMOTE := #Init, L_SIM :=, L_RESET := #Reset, AUT_OP :=, MAN_OP :=, SIM_OP :=, FB_OPEN :=, FB_CLOSE :=, L_MON := #Init, MON_T :=, MON_T_CLOSE :=, INSTANCE := 'AV-14.01', RESTART :=, VISIBILITY :=, OPdwCmd :=, QdwState =>, QwState =>, QCLOSING =>, QCLOSE =>, QOPENING =>, QOPEN =>, QCMD_OP => "AV-14.01", QMON =>, QMON_ERR =>, QMON_T =>, QMON_T_CLOSE =>, QMAN_AUT =>, QREMOTE =>, QSIM =>, QLOCK =>, QERR =>, QERR_EXT =>, QwAlarm =>)
   END_RUNG
   // the same network as SCL:
   #"AV-14.01"(LOCK := #lock,   // "Valve"
               LIOP_SEL := #Init,
               L_AUT := #Init,
               L_REMOTE := #Init,
               L_RESET := #Reset,
               L_MON := #Init,
               INSTANCE := 'AV-14.01',
               QCMD_OP => "AV-14.01");
END_REGION

REGION Network 24: AV-14.02 w ZSC
   RUNG wire#powerrail
      #"AV-14.02"(LOCK :=, ERR_EXTERN :=, LIOP_SEL := #Init, L_AUT := #Init, L_REMOTE := #Init, L_SIM :=, L_RESET := #Reset, AUT_OP :=, MAN_OP :=, SIM_OP :=, FB_OPEN :=, FB_CLOSE :=, L_MON := #Init, MON_T :=, MON_T_CLOSE :=, INSTANCE := 'AV-14.02', RESTART :=, VISIBILITY :=, OPdwCmd :=, QdwState =>, QwState =>, QCLOSING =>, QCLOSE =>, QOPENING =>, QOPEN =>, QCMD_OP => "AV-14.02", QMON =>, QMON_ERR =>, QMON_T =>, QMON_T_CLOSE =>, QMAN_AUT =>, QREMOTE =>, QSIM =>, QLOCK =>, QERR =>, QERR_EXT =>, QwAlarm =>)
   END_RUNG
   // the same network as SCL:
   #"AV-14.02"(LIOP_SEL := #Init,   // "Valve"
               L_AUT := #Init,
               L_REMOTE := #Init,
               L_RESET := #Reset,
               L_MON := #Init,
               INSTANCE := 'AV-14.02',
               QCMD_OP => "AV-14.02");
END_REGION

REGION Network 25: AV-14.03
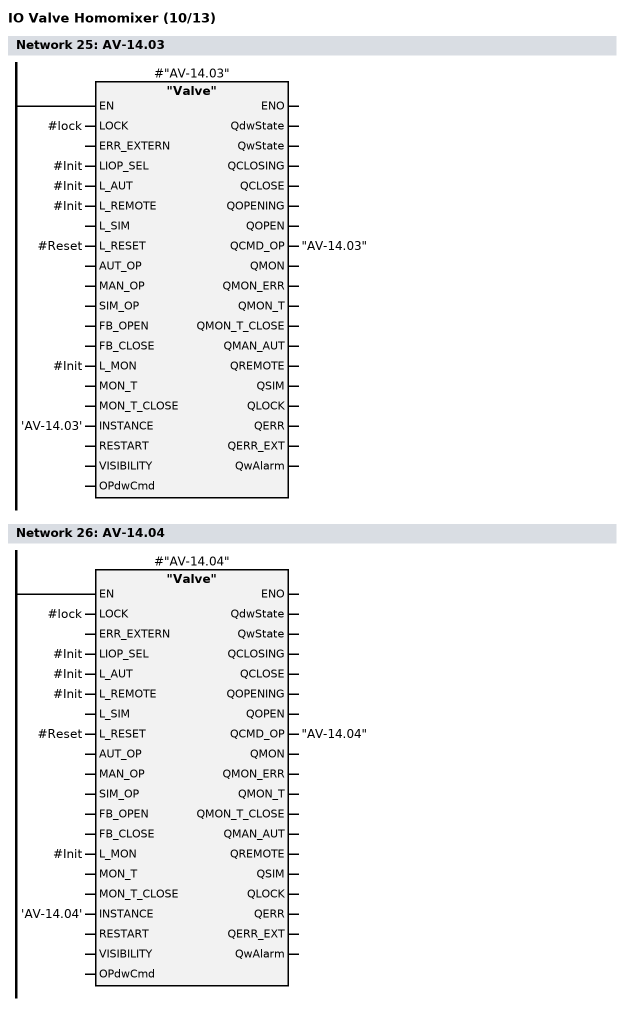
   RUNG wire#powerrail
      #"AV-14.03"(LOCK := #lock, ERR_EXTERN :=, LIOP_SEL := #Init, L_AUT := #Init, L_REMOTE := #Init, L_SIM :=, L_RESET := #Reset, AUT_OP :=, MAN_OP :=, SIM_OP :=, FB_OPEN :=, FB_CLOSE :=, L_MON := #Init, MON_T :=, MON_T_CLOSE :=, INSTANCE := 'AV-14.03', RESTART :=, VISIBILITY :=, OPdwCmd :=, QdwState =>, QwState =>, QCLOSING =>, QCLOSE =>, QOPENING =>, QOPEN =>, QCMD_OP => "AV-14.03", QMON =>, QMON_ERR =>, QMON_T =>, QMON_T_CLOSE =>, QMAN_AUT =>, QREMOTE =>, QSIM =>, QLOCK =>, QERR =>, QERR_EXT =>, QwAlarm =>)
   END_RUNG
   // the same network as SCL:
   #"AV-14.03"(LOCK := #lock,   // "Valve"
               LIOP_SEL := #Init,
               L_AUT := #Init,
               L_REMOTE := #Init,
               L_RESET := #Reset,
               L_MON := #Init,
               INSTANCE := 'AV-14.03',
               QCMD_OP => "AV-14.03");
END_REGION

REGION Network 26: AV-14.04
   RUNG wire#powerrail
      #"AV-14.04"(LOCK := #lock, ERR_EXTERN :=, LIOP_SEL := #Init, L_AUT := #Init, L_REMOTE := #Init, L_SIM :=, L_RESET := #Reset, AUT_OP :=, MAN_OP :=, SIM_OP :=, FB_OPEN :=, FB_CLOSE :=, L_MON := #Init, MON_T :=, MON_T_CLOSE :=, INSTANCE := 'AV-14.04', RESTART :=, VISIBILITY :=, OPdwCmd :=, QdwState =>, QwState =>, QCLOSING =>, QCLOSE =>, QOPENING =>, QOPEN =>, QCMD_OP => "AV-14.04", QMON =>, QMON_ERR =>, QMON_T =>, QMON_T_CLOSE =>, QMAN_AUT =>, QREMOTE =>, QSIM =>, QLOCK =>, QERR =>, QERR_EXT =>, QwAlarm =>)
   END_RUNG
   // the same network as SCL:
   #"AV-14.04"(LOCK := #lock,   // "Valve"
               LIOP_SEL := #Init,
               L_AUT := #Init,
               L_REMOTE := #Init,
               L_RESET := #Reset,
               L_MON := #Init,
               INSTANCE := 'AV-14.04',
               QCMD_OP => "AV-14.04");
END_REGION

REGION Network 27: AV-14.05
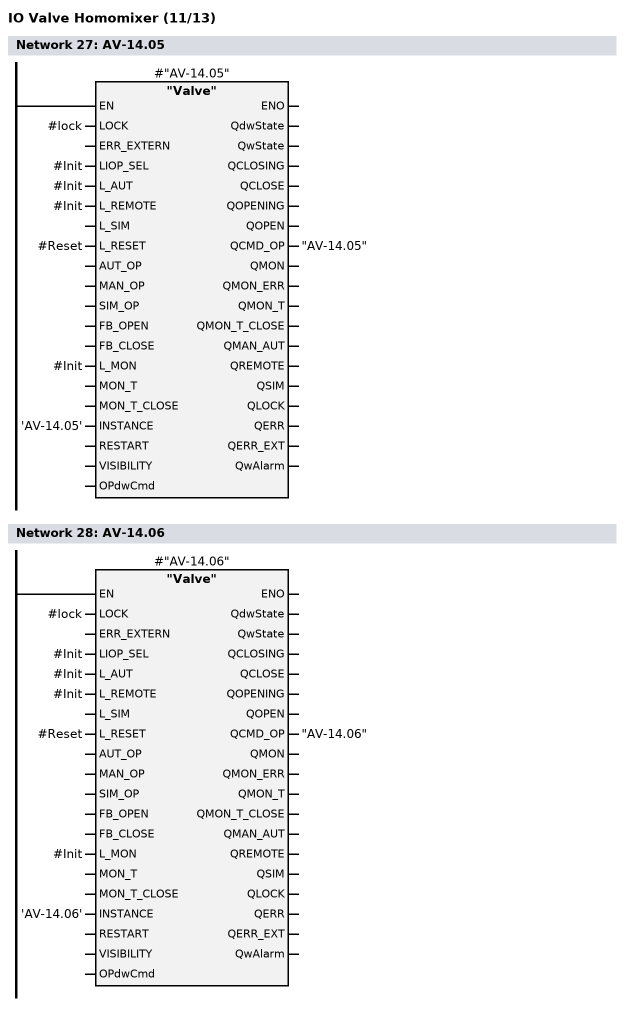
   RUNG wire#powerrail
      #"AV-14.05"(LOCK := #lock, ERR_EXTERN :=, LIOP_SEL := #Init, L_AUT := #Init, L_REMOTE := #Init, L_SIM :=, L_RESET := #Reset, AUT_OP :=, MAN_OP :=, SIM_OP :=, FB_OPEN :=, FB_CLOSE :=, L_MON := #Init, MON_T :=, MON_T_CLOSE :=, INSTANCE := 'AV-14.05', RESTART :=, VISIBILITY :=, OPdwCmd :=, QdwState =>, QwState =>, QCLOSING =>, QCLOSE =>, QOPENING =>, QOPEN =>, QCMD_OP => "AV-14.05", QMON =>, QMON_ERR =>, QMON_T =>, QMON_T_CLOSE =>, QMAN_AUT =>, QREMOTE =>, QSIM =>, QLOCK =>, QERR =>, QERR_EXT =>, QwAlarm =>)
   END_RUNG
   // the same network as SCL:
   #"AV-14.05"(LOCK := #lock,   // "Valve"
               LIOP_SEL := #Init,
               L_AUT := #Init,
               L_REMOTE := #Init,
               L_RESET := #Reset,
               L_MON := #Init,
               INSTANCE := 'AV-14.05',
               QCMD_OP => "AV-14.05");
END_REGION

REGION Network 28: AV-14.06
   RUNG wire#powerrail
      #"AV-14.06"(LOCK := #lock, ERR_EXTERN :=, LIOP_SEL := #Init, L_AUT := #Init, L_REMOTE := #Init, L_SIM :=, L_RESET := #Reset, AUT_OP :=, MAN_OP :=, SIM_OP :=, FB_OPEN :=, FB_CLOSE :=, L_MON := #Init, MON_T :=, MON_T_CLOSE :=, INSTANCE := 'AV-14.06', RESTART :=, VISIBILITY :=, OPdwCmd :=, QdwState =>, QwState =>, QCLOSING =>, QCLOSE =>, QOPENING =>, QOPEN =>, QCMD_OP => "AV-14.06", QMON =>, QMON_ERR =>, QMON_T =>, QMON_T_CLOSE =>, QMAN_AUT =>, QREMOTE =>, QSIM =>, QLOCK =>, QERR =>, QERR_EXT =>, QwAlarm =>)
   END_RUNG
   // the same network as SCL:
   #"AV-14.06"(LOCK := #lock,   // "Valve"
               LIOP_SEL := #Init,
               L_AUT := #Init,
               L_REMOTE := #Init,
               L_RESET := #Reset,
               L_MON := #Init,
               INSTANCE := 'AV-14.06',
               QCMD_OP => "AV-14.06");
END_REGION

REGION Network 29: AV-14.07
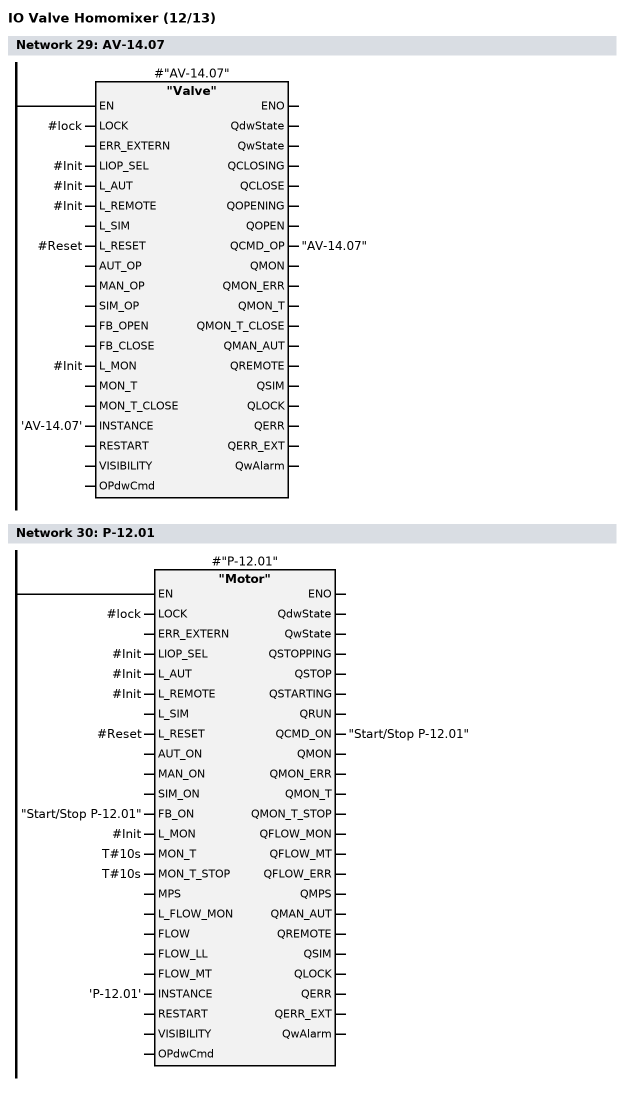
   RUNG wire#powerrail
      #"AV-14.07"(LOCK := #lock, ERR_EXTERN :=, LIOP_SEL := #Init, L_AUT := #Init, L_REMOTE := #Init, L_SIM :=, L_RESET := #Reset, AUT_OP :=, MAN_OP :=, SIM_OP :=, FB_OPEN :=, FB_CLOSE :=, L_MON := #Init, MON_T :=, MON_T_CLOSE :=, INSTANCE := 'AV-14.07', RESTART :=, VISIBILITY :=, OPdwCmd :=, QdwState =>, QwState =>, QCLOSING =>, QCLOSE =>, QOPENING =>, QOPEN =>, QCMD_OP => "AV-14.07", QMON =>, QMON_ERR =>, QMON_T =>, QMON_T_CLOSE =>, QMAN_AUT =>, QREMOTE =>, QSIM =>, QLOCK =>, QERR =>, QERR_EXT =>, QwAlarm =>)
   END_RUNG
   // the same network as SCL:
   #"AV-14.07"(LOCK := #lock,   // "Valve"
               LIOP_SEL := #Init,
               L_AUT := #Init,
               L_REMOTE := #Init,
               L_RESET := #Reset,
               L_MON := #Init,
               INSTANCE := 'AV-14.07',
               QCMD_OP => "AV-14.07");
END_REGION

REGION Network 30: P-12.01
   RUNG wire#powerrail
      #"P-12.01"(LOCK := #lock, ERR_EXTERN :=, LIOP_SEL := #Init, L_AUT := #Init, L_REMOTE := #Init, L_SIM :=, L_RESET := #Reset, AUT_ON :=, MAN_ON :=, SIM_ON :=, FB_ON := "Start/Stop P-12.01", L_MON := #Init, MON_T := T#10s, MON_T_STOP := T#10s, MPS :=, L_FLOW_MON :=, FLOW :=, FLOW_LL :=, FLOW_MT :=, INSTANCE := 'P-12.01', RESTART :=, VISIBILITY :=, OPdwCmd :=, QdwState =>, QwState =>, QSTOPPING =>, QSTOP =>, QSTARTING =>, QRUN =>, QCMD_ON => "Start/Stop P-12.01", QMON =>, QMON_ERR =>, QMON_T =>, QMON_T_STOP =>, QFLOW_MON =>, QFLOW_MT =>, QFLOW_ERR =>, QMPS =>, QMAN_AUT =>, QREMOTE =>, QSIM =>, QLOCK =>, QERR =>, QERR_EXT =>, QwAlarm =>)
   END_RUNG
   // the same network as SCL:
   #"P-12.01"(LOCK := #lock,   // "Motor"
              LIOP_SEL := #Init,
              L_AUT := #Init,
              L_REMOTE := #Init,
              L_RESET := #Reset,
              FB_ON := "Start/Stop P-12.01",
              L_MON := #Init,
              MON_T := T#10s,
              MON_T_STOP := T#10s,
              INSTANCE := 'P-12.01',
              QCMD_ON => "Start/Stop P-12.01");
END_REGION

REGION Network 31: P-13.01
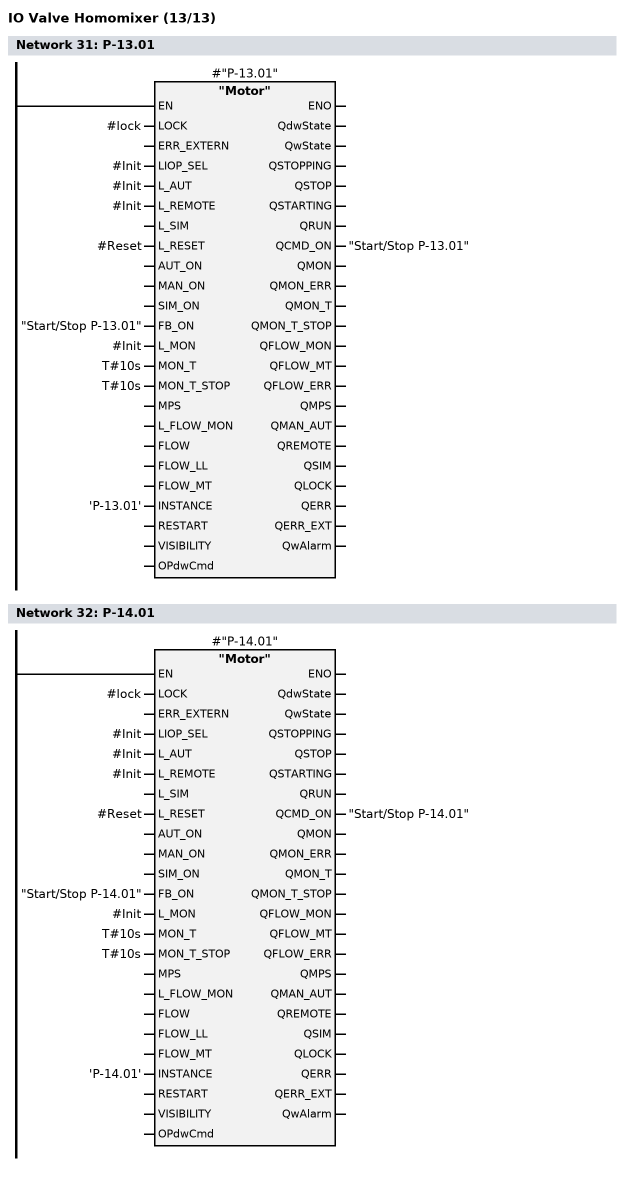
   RUNG wire#powerrail
      #"P-13.01"(LOCK := #lock, ERR_EXTERN :=, LIOP_SEL := #Init, L_AUT := #Init, L_REMOTE := #Init, L_SIM :=, L_RESET := #Reset, AUT_ON :=, MAN_ON :=, SIM_ON :=, FB_ON := "Start/Stop P-13.01", L_MON := #Init, MON_T := T#10s, MON_T_STOP := T#10s, MPS :=, L_FLOW_MON :=, FLOW :=, FLOW_LL :=, FLOW_MT :=, INSTANCE := 'P-13.01', RESTART :=, VISIBILITY :=, OPdwCmd :=, QdwState =>, QwState =>, QSTOPPING =>, QSTOP =>, QSTARTING =>, QRUN =>, QCMD_ON => "Start/Stop P-13.01", QMON =>, QMON_ERR =>, QMON_T =>, QMON_T_STOP =>, QFLOW_MON =>, QFLOW_MT =>, QFLOW_ERR =>, QMPS =>, QMAN_AUT =>, QREMOTE =>, QSIM =>, QLOCK =>, QERR =>, QERR_EXT =>, QwAlarm =>)
   END_RUNG
   // the same network as SCL:
   #"P-13.01"(LOCK := #lock,   // "Motor"
              LIOP_SEL := #Init,
              L_AUT := #Init,
              L_REMOTE := #Init,
              L_RESET := #Reset,
              FB_ON := "Start/Stop P-13.01",
              L_MON := #Init,
              MON_T := T#10s,
              MON_T_STOP := T#10s,
              INSTANCE := 'P-13.01',
              QCMD_ON => "Start/Stop P-13.01");
END_REGION

REGION Network 32: P-14.01
   RUNG wire#powerrail
      #"P-14.01"(LOCK := #lock, ERR_EXTERN :=, LIOP_SEL := #Init, L_AUT := #Init, L_REMOTE := #Init, L_SIM :=, L_RESET := #Reset, AUT_ON :=, MAN_ON :=, SIM_ON :=, FB_ON := "Start/Stop P-14.01", L_MON := #Init, MON_T := T#10s, MON_T_STOP := T#10s, MPS :=, L_FLOW_MON :=, FLOW :=, FLOW_LL :=, FLOW_MT :=, INSTANCE := 'P-14.01', RESTART :=, VISIBILITY :=, OPdwCmd :=, QdwState =>, QwState =>, QSTOPPING =>, QSTOP =>, QSTARTING =>, QRUN =>, QCMD_ON => "Start/Stop P-14.01", QMON =>, QMON_ERR =>, QMON_T =>, QMON_T_STOP =>, QFLOW_MON =>, QFLOW_MT =>, QFLOW_ERR =>, QMPS =>, QMAN_AUT =>, QREMOTE =>, QSIM =>, QLOCK =>, QERR =>, QERR_EXT =>, QwAlarm =>)
   END_RUNG
   // the same network as SCL:
   #"P-14.01"(LOCK := #lock,   // "Motor"
              LIOP_SEL := #Init,
              L_AUT := #Init,
              L_REMOTE := #Init,
              L_RESET := #Reset,
              FB_ON := "Start/Stop P-14.01",
              L_MON := #Init,
              MON_T := T#10s,
              MON_T_STOP := T#10s,
              INSTANCE := 'P-14.01',
              QCMD_ON => "Start/Stop P-14.01");
END_REGION
END_FUNCTION_BLOCK

FUNCTION "Pulse" : Void   // FC10, LAD
{ S7_Optimized_Access := 'TRUE' }
VERSION : 0.1
// stored: AutoNumber true, IsIECCheckEnabled false, SetENOAutomatically false, UDAEnableTagReadback false
   VAR_TEMP   // added for the SCL form of the ladder/FBD networks
      _w1 : Bool;
      _s5time1 : S5Time;
      _w2 : Bool;
      _s5time2 : S5Time;
   END_VAR
BEGIN

REGION Network 1: Timer 5s/ 1M
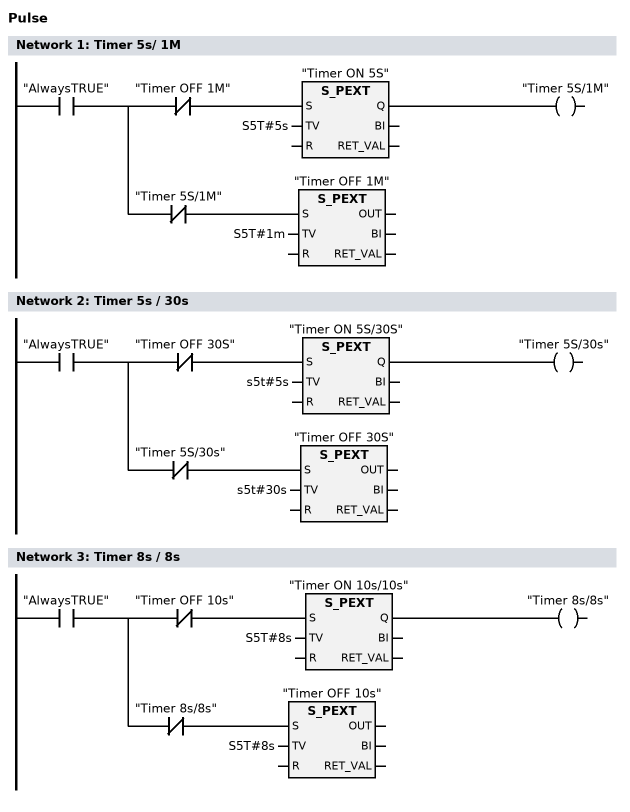
   RUNG wire#powerrail
      Contact( "AlwaysTRUE" )
      wire#w1
      I_Contact( "Timer OFF 1M" )
      S_PEXT(T_NO := "Timer ON 5S", TV := S5T#5s, R :=, BI =>, RET_VAL =>)
      Coil( "Timer 5S/1M" )
   END_RUNG
   RUNG wire#w1
      I_Contact( "Timer 5S/1M" )
      S_PEXT(T_NO := "Timer OFF 1M", TV := S5T#1m, R :=, BI =>, RET_VAL =>)
   END_RUNG
   // the same network as SCL:
   #_w2 := "AlwaysTRUE";
   #_s5time1 := S_PEXT(T_NO := "Timer ON 5S", S := "AlwaysTRUE" AND NOT "Timer OFF 1M", TV := S5T#5s, Q => #_w1);
   "Timer 5S/1M" := #_w1;
   #_s5time2 := S_PEXT(T_NO := "Timer OFF 1M", S := #_w2 AND NOT "Timer 5S/1M", TV := S5T#1m);
END_REGION

REGION Network 2: Timer 5s / 30s
   RUNG wire#powerrail
      Contact( "AlwaysTRUE" )
      wire#w1
      I_Contact( "Timer OFF 30S" )
      S_PEXT(T_NO := "Timer ON 5S/30S", TV := s5t#5s, R :=, BI =>, RET_VAL =>)
      Coil( "Timer 5S/30s" )
   END_RUNG
   RUNG wire#w1
      I_Contact( "Timer 5S/30s" )
      S_PEXT(T_NO := "Timer OFF 30S", TV := s5t#30s, R :=, BI =>, RET_VAL =>)
   END_RUNG
   // the same network as SCL:
   #_w2 := "AlwaysTRUE";
   #_s5time1 := S_PEXT(T_NO := "Timer ON 5S/30S",
                       S := "AlwaysTRUE" AND NOT "Timer OFF 30S",
                       TV := s5t#5s,
                       Q => #_w1);
   "Timer 5S/30s" := #_w1;
   #_s5time2 := S_PEXT(T_NO := "Timer OFF 30S", S := #_w2 AND NOT "Timer 5S/30s", TV := s5t#30s);
END_REGION

REGION Network 3: Timer 8s / 8s
   RUNG wire#powerrail
      Contact( "AlwaysTRUE" )
      wire#w1
      I_Contact( "Timer OFF 10s" )
      S_PEXT(T_NO := "Timer ON 10s/10s", TV := S5T#8s, R :=, BI =>, RET_VAL =>)
      Coil( "Timer 8s/8s" )
   END_RUNG
   RUNG wire#w1
      I_Contact( "Timer 8s/8s" )
      S_PEXT(T_NO := "Timer OFF 10s", TV := S5T#8s, R :=, BI =>, RET_VAL =>)
   END_RUNG
   // the same network as SCL:
   #_w2 := "AlwaysTRUE";
   #_s5time1 := S_PEXT(T_NO := "Timer ON 10s/10s",
                       S := "AlwaysTRUE" AND NOT "Timer OFF 10s",
                       TV := S5T#8s,
                       Q => #_w1);
   "Timer 8s/8s" := #_w1;
   #_s5time2 := S_PEXT(T_NO := "Timer OFF 10s", S := #_w2 AND NOT "Timer 8s/8s", TV := S5T#8s);
END_REGION
END_FUNCTION

FUNCTION "BlendingArea" : Void   // FC201, LAD
{ S7_Optimized_Access := 'TRUE' }
VERSION : 0.1
// stored: AutoNumber false, IsIECCheckEnabled false, SetENOAutomatically false, UDAEnableTagReadback false
   VAR_TEMP   // added for the SCL form of the ladder/FBD networks
      _w1 : Bool;
      _w2 : Bool;
   END_VAR
BEGIN

REGION Network 1: Analog
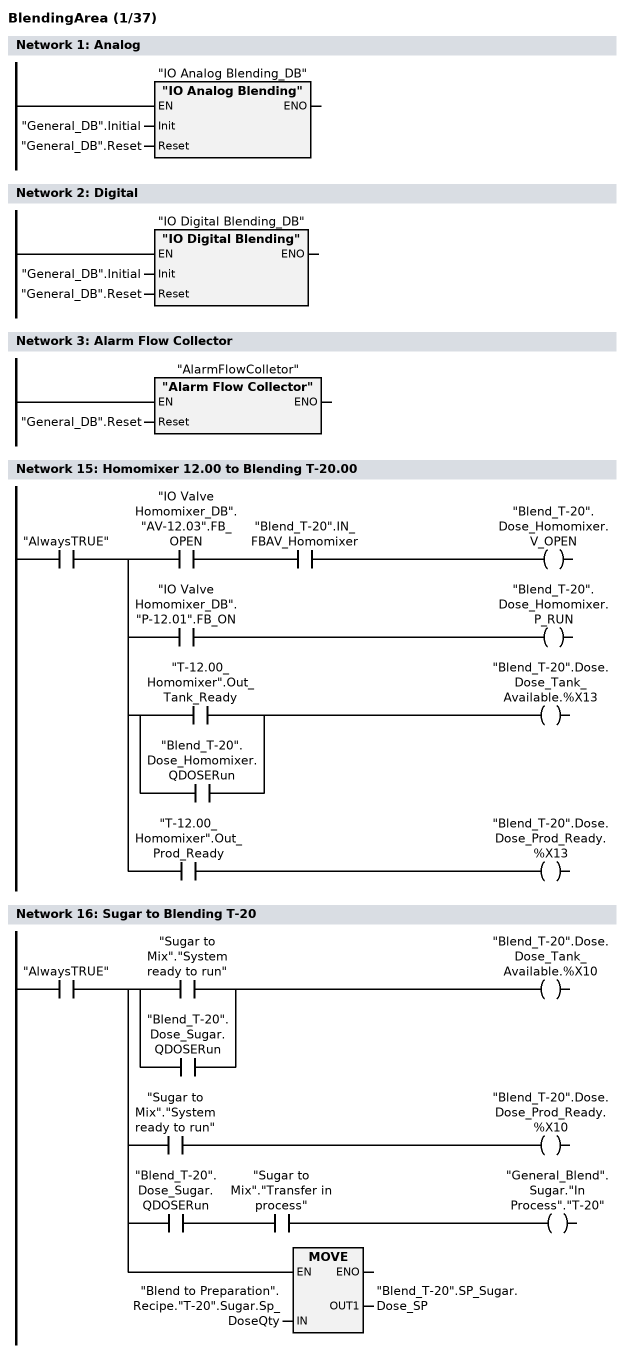
   RUNG wire#powerrail
      "IO Analog Blending_DB"(Init := "General_DB".Initial, Reset := "General_DB".Reset)
   END_RUNG
   // the same network as SCL:
   "IO Analog Blending_DB"(Init := "General_DB".Initial, Reset := "General_DB".Reset);   // "IO Analog Blending"
END_REGION

REGION Network 2: Digital
   RUNG wire#powerrail
      "IO Digital Blending_DB"(Init := "General_DB".Initial, Reset := "General_DB".Reset)
   END_RUNG
   // the same network as SCL:
   "IO Digital Blending_DB"(Init := "General_DB".Initial, Reset := "General_DB".Reset);   // "IO Digital Blending"
END_REGION

REGION Network 3: Alarm Flow Collector
   RUNG wire#powerrail
      "AlarmFlowColletor"(Reset := "General_DB".Reset)
   END_RUNG
   // the same network as SCL:
   "AlarmFlowColletor"(Reset := "General_DB".Reset);   // "Alarm Flow Collector"
END_REGION

NETWORK
TITLE = ChiliAwetan1 to Blending T-20
//Valve Open
      A     "Preparation to Blend"."T-02_ChiliAwetan_1".Valve_Open;
      A(;
      O(;
      A     "Blend_T-20".Dose.Dose_Header_Req.%X0;
      A     "Blend_T-20".IN_FBAV_Header1;
      );
      O(;
      A     "Blend_T-20".Dose.Dose_Header_Req.%X16;
      A     "Blend_T-20".IN_FBAV_Header2;
      );
      );
      =     "Blend_T-20".Dose_ChiliAwetan1.V_OPEN;
//Pump On
      O     "Preparation to Blend"."T-02_ChiliAwetan_1".Pump_Run;
      =     "Blend_T-20".Dose_ChiliAwetan1.P_RUN;
//Tank Available
      O     "Preparation to Blend"."T-02_ChiliAwetan_1".Tank_Available;
      O     "Blend_T-20".Dose_ChiliAwetan1.QDOSERun;
      =     "Blend_T-20".Dose.Dose_Tank_Available.%X0;
//Product Ready
      O     "Preparation to Blend"."T-02_ChiliAwetan_1".Product_Ready;
      =     "Blend_T-20".Dose.Dose_Prod_Ready.%X0;
//Level Tank
      L     "Preparation to Blend"."T-02_ChiliAwetan_1".Level;
      T     "Blend_T-20"."Dose_Level_%"."ChiliAwetan1%";


NETWORK
TITLE = ChiliAwetan2 to Blending T-20
//Valve Open
      A     "Preparation to Blend"."T-03_ChiliAwetan_2".Valve_Open;
      A(;
      O(;
      A     "Blend_T-20".Dose.Dose_Header_Req.%X1;
      A     "Blend_T-20".IN_FBAV_Header1;
      );
      O(;
      A     "Blend_T-20".Dose.Dose_Header_Req.%X17;
      A     "Blend_T-20".IN_FBAV_Header2;
      );
      );
      =     "Blend_T-20".Dose_ChiliAwetan2.V_OPEN;
//Pump On
      O     "Preparation to Blend"."T-03_ChiliAwetan_2".Pump_Run;
      =     "Blend_T-20".Dose_ChiliAwetan2.P_RUN;
//Tank Available
      O     "Preparation to Blend"."T-03_ChiliAwetan_2".Tank_Available;
      O     "Blend_T-20".Dose_ChiliAwetan2.QDOSERun;
      =     "Blend_T-20".Dose.Dose_Tank_Available.%X1;
//Product Ready
      O     "Preparation to Blend"."T-03_ChiliAwetan_2".Product_Ready;
      =     "Blend_T-20".Dose.Dose_Prod_Ready.%X1;
//Level Tank
      L     "Preparation to Blend"."T-03_ChiliAwetan_2".Level;
      T     "Blend_T-20"."Dose_Level_%"."ChiliAwetan2%";


NETWORK
TITLE = ChiliAwetan3 to Blending T-20
//Valve Open
      A     "Preparation to Blend"."T-04_ChiliAwetan_3".Valve_Open;
      A(;
      O(;
      A     "Blend_T-20".Dose.Dose_Header_Req.%X2;
      A     "Blend_T-20".IN_FBAV_Header1;
      );
      O(;
      A     "Blend_T-20".Dose.Dose_Header_Req.%X18;
      A     "Blend_T-20".IN_FBAV_Header2;
      );
      );
      =     "Blend_T-20".Dose_ChiliAwetan3.V_OPEN;
//Pump On
      O     "Preparation to Blend"."T-04_ChiliAwetan_3".Pump_Run;
      =     "Blend_T-20".Dose_ChiliAwetan3.P_RUN;
//Tank Available
      O     "Preparation to Blend"."T-04_ChiliAwetan_3".Tank_Available;
      O     "Blend_T-20".Dose_ChiliAwetan3.QDOSERun;
      =     "Blend_T-20".Dose.Dose_Tank_Available.%X2;
//Product Ready
      O     "Preparation to Blend"."T-04_ChiliAwetan_3".Product_Ready;
      =     "Blend_T-20".Dose.Dose_Prod_Ready.%X2;
//Level Tank
      L     "Preparation to Blend"."T-04_ChiliAwetan_3".Level;
      T     "Blend_T-20"."Dose_Level_%"."ChiliAwetan3%";


NETWORK
TITLE = Tomato to Blending T-20
//Valve Open
      A     "Preparation to Blend"."T-05_Tomato".Valve_Open;
      A(;
      O(;
      A     "Blend_T-20".Dose.Dose_Header_Req.%X3;
      A     "Blend_T-20".IN_FBAV_Header1;
      );
      O(;
      A     "Blend_T-20".Dose.Dose_Header_Req.%X19;
      A     "Blend_T-20".IN_FBAV_Header2;
      );
      );
      =     "Blend_T-20".Dose_Tomato.V_OPEN;
//Pump On
      O     "Preparation to Blend"."T-05_Tomato".Pump_Run;
      =     "Blend_T-20".Dose_Tomato.P_RUN;
//Tank Available
      O     "Preparation to Blend"."T-05_Tomato".Tank_Available;
      O     "Blend_T-20".Dose_Tomato.QDOSERun;
      =     "Blend_T-20".Dose.Dose_Tank_Available.%X3;
//Product Ready
      O     "Preparation to Blend"."T-05_Tomato".Product_Ready;
      =     "Blend_T-20".Dose.Dose_Prod_Ready.%X3;
//Level Tank
      L     "Preparation to Blend"."T-05_Tomato".Level;
      T     "Blend_T-20"."Dose_Level_%"."Tomato%";


NETWORK
TITLE = ChiliFresh1 to Blending T-20
//Valve Open
      A     "Preparation to Blend"."T-06_ChiliFresh_1".Valve_Open;
      A(;
      O(;
      A     "Blend_T-20".Dose.Dose_Header_Req.%X4;
      A     "Blend_T-20".IN_FBAV_Header1;
      );
      O(;
      A     "Blend_T-20".Dose.Dose_Header_Req.%X20;
      A     "Blend_T-20".IN_FBAV_Header2;
      );
      );
      =     "Blend_T-20".Dose_ChiliFresh1.V_OPEN;
//Pump On
      O     "Preparation to Blend"."T-06_ChiliFresh_1".Pump_Run;
      =     "Blend_T-20".Dose_ChiliFresh1.P_RUN;
//Tank Available
      O     "Preparation to Blend"."T-06_ChiliFresh_1".Tank_Available;
      O     "Blend_T-20".Dose_ChiliFresh1.QDOSERun;
      =     "Blend_T-20".Dose.Dose_Tank_Available.%X4;
//Product Ready
      O     "Preparation to Blend"."T-06_ChiliFresh_1".Product_Ready;
      =     "Blend_T-20".Dose.Dose_Prod_Ready.%X4;
//Level Tank
      L     "Preparation to Blend"."T-06_ChiliFresh_1".Level;
      T     "Blend_T-20"."Dose_Level_%"."ChiliFresh1%";


NETWORK
TITLE = ChiliFresh2 to Blending T-20
//Valve Open
      A     "Preparation to Blend"."T-07_ChiliFresh_2".Valve_Open;
      A(;
      O(;
      A     "Blend_T-20".Dose.Dose_Header_Req.%X5;
      A     "Blend_T-20".IN_FBAV_Header1;
      );
      O(;
      A     "Blend_T-20".Dose.Dose_Header_Req.%X21;
      A     "Blend_T-20".IN_FBAV_Header2;
      );
      );
      =     "Blend_T-20".Dose_ChiliFresh2.V_OPEN;
//Pump On
      O     "Preparation to Blend"."T-07_ChiliFresh_2".Pump_Run;
      =     "Blend_T-20".Dose_ChiliFresh2.P_RUN;
//Tank Available
      O     "Preparation to Blend"."T-07_ChiliFresh_2".Tank_Available;
      O     "Blend_T-20".Dose_ChiliFresh2.QDOSERun;
      =     "Blend_T-20".Dose.Dose_Tank_Available.%X5;
//Product Ready
      O     "Preparation to Blend"."T-07_ChiliFresh_2".Product_Ready;
      =     "Blend_T-20".Dose.Dose_Prod_Ready.%X5;
//Level Tank
      L     "Preparation to Blend"."T-07_ChiliFresh_2".Level;
      T     "Blend_T-20"."Dose_Level_%"."ChiliFresh2%";


NETWORK
TITLE = ChiliFresh3 to Blending T-20
//Valve Open
      A     "Preparation to Blend"."T-08_ChiliFresh_3".Valve_Open;
      A(;
      O(;
      A     "Blend_T-20".Dose.Dose_Header_Req.%X6;
      A     "Blend_T-20".IN_FBAV_Header1;
      );
      O(;
      A     "Blend_T-20".Dose.Dose_Header_Req.%X22;
      A     "Blend_T-20".IN_FBAV_Header2;
      );
      );
      =     "Blend_T-20".Dose_ChiliFresh3.V_OPEN;
//Pump On
      O     "Preparation to Blend"."T-08_ChiliFresh_3".Pump_Run;
      =     "Blend_T-20".Dose_ChiliFresh3.P_RUN;
//Tank Available
      O     "Preparation to Blend"."T-08_ChiliFresh_3".Tank_Available;
      O     "Blend_T-20".Dose_ChiliFresh3.QDOSERun;
      =     "Blend_T-20".Dose.Dose_Tank_Available.%X6;
//Product Ready
      O     "Preparation to Blend"."T-08_ChiliFresh_3".Product_Ready;
      =     "Blend_T-20".Dose.Dose_Prod_Ready.%X6;
//Level Tank
      L     "Preparation to Blend"."T-08_ChiliFresh_3".Level;
      T     "Blend_T-20"."Dose_Level_%"."ChiliFresh3%";


NETWORK
TITLE = Garlic to Blending T-20
//Valve Open
      A     "Preparation to Blend"."T-09_Garlic".Valve_Open;
      A(;
      O(;
      A     "Blend_T-20".Dose.Dose_Header_Req.%X7;
      A     "Blend_T-20".IN_FBAV_Header1;
      );
      O(;
      A     "Blend_T-20".Dose.Dose_Header_Req.%X23;
      A     "Blend_T-20".IN_FBAV_Header2;
      );
      );
      =     "Blend_T-20".Dose_Garlic.V_OPEN;
//Pump On
      O     "Preparation to Blend"."T-09_Garlic".Pump_Run;
      =     "Blend_T-20".Dose_Garlic.P_RUN;
//Tank Available
      O     "Preparation to Blend"."T-09_Garlic".Tank_Available;
      O     "Blend_T-20".Dose_Garlic.QDOSERun;
      =     "Blend_T-20".Dose.Dose_Tank_Available.%X7;
//Product Ready
      O     "Preparation to Blend"."T-09_Garlic".Product_Ready;
      =     "Blend_T-20".Dose.Dose_Prod_Ready.%X7;
//Level Tank
      L     "Preparation to Blend"."T-09_Garlic".Level;
      T     "Blend_T-20"."Dose_Level_%"."Garlic%";


NETWORK
TITLE = Vinegar to Blending T-20
//Valve Open
      A     "Preparation to Blend"."T-10_Vinegar".Valve_Open;
      A     "Blend_T-20".IN_FBAV_Vinegar;
      =     "Blend_T-20".Dose_Vinegar.V_OPEN;
//Pump On
      O     "Preparation to Blend"."T-10_Vinegar".Pump_Run;
      =     "Blend_T-20".Dose_Vinegar.P_RUN;
//Tank Available
      O     "Preparation to Blend"."T-10_Vinegar".Tank_Available;
      O     "Blend_T-20".Dose_Vinegar.QDOSERun;
      =     "Blend_T-20".Dose.Dose_Tank_Available.%X9;
//Product Ready
      O     "Preparation to Blend"."T-10_Vinegar".Product_Ready;
      =     "Blend_T-20".Dose.Dose_Prod_Ready.%X9;
//Level Tank
      L     "Preparation to Blend"."T-10_Vinegar".Level;
      T     "Blend_T-20"."Dose_Level_%"."Vinegar%";


NETWORK
TITLE = HW to Blending T-20
//Valve Open
      A     "Preparation to Blend"."T-51_HW".Valve_Open;
      A(;
      O(;
      A     "Blend_T-20".Dose.Dose_Header_Req.%X8;
      A     "Blend_T-20".IN_FBAV_Header1;
      );
      O(;
      A     "Blend_T-20".Dose.Dose_Header_Req.%X24;
      A     "Blend_T-20".IN_FBAV_Header2;
      );
      );
      =     "Blend_T-20".Dose_HW.V_OPEN;
//Pump On
      O     "Preparation to Blend"."T-51_HW".Pump_Run;
      =     "Blend_T-20".Dose_HW.P_RUN;
//Tank Available
      O     "Preparation to Blend"."T-51_HW".Tank_Available;
      O     "Blend_T-20".Dose_HW.QDOSERun;
      =     "Blend_T-20".Dose.Dose_Tank_Available.%X8;
//Product Ready
      O     "Preparation to Blend"."T-51_HW".Product_Ready;
      =     "Blend_T-20".Dose.Dose_Prod_Ready.%X8;
//Level Tank
// L     "Preparation to Blend"."T-01_HW".Level
// T     "Blend_T-20"."Dose_Level_%"."HW%"


REGION Network 15: Homomixer 12.00 to Blending T-20.00
   RUNG wire#powerrail
      Contact( "AlwaysTRUE" )
      wire#w1
      Contact( "IO Valve Homomixer_DB"."AV-12.03".FB_OPEN )
      Contact( "Blend_T-20".IN_FBAV_Homomixer )
      Coil( "Blend_T-20".Dose_Homomixer.V_OPEN )
   END_RUNG
   RUNG wire#w1
      Contact( "IO Valve Homomixer_DB"."P-12.01".FB_ON )
      Coil( "Blend_T-20".Dose_Homomixer.P_RUN )
   END_RUNG
   RUNG wire#w1
      Contact( "T-12.00_Homomixer".Out_Tank_Ready )
      wire#w2
      Coil( "Blend_T-20".Dose.Dose_Tank_Available.%X13 )
   END_RUNG
   RUNG wire#w1
      Contact( "Blend_T-20".Dose_Homomixer.QDOSERun )
   END_RUNG wire#w2
   RUNG wire#w1
      Contact( "T-12.00_Homomixer".Out_Prod_Ready )
      Coil( "Blend_T-20".Dose.Dose_Prod_Ready.%X13 )
   END_RUNG
   // the same network as SCL:
   "Blend_T-20".Dose_Homomixer.V_OPEN := "AlwaysTRUE" AND "IO Valve Homomixer_DB"."AV-12.03".FB_OPEN AND "Blend_T-20".IN_FBAV_Homomixer;
   "Blend_T-20".Dose_Homomixer.P_RUN := "AlwaysTRUE" AND "IO Valve Homomixer_DB"."P-12.01".FB_ON;
   "Blend_T-20".Dose.Dose_Tank_Available.%X13 := "AlwaysTRUE" AND ("T-12.00_Homomixer".Out_Tank_Ready OR "Blend_T-20".Dose_Homomixer.QDOSERun);
   "Blend_T-20".Dose.Dose_Prod_Ready.%X13 := "AlwaysTRUE" AND "T-12.00_Homomixer".Out_Prod_Ready;
END_REGION

REGION Network 16: Sugar to Blending T-20
   RUNG wire#powerrail
      Contact( "AlwaysTRUE" )
      wire#w1
      Contact( "Sugar to Mix"."System ready to run" )
      wire#w2
      Coil( "Blend_T-20".Dose.Dose_Tank_Available.%X10 )
   END_RUNG
   RUNG wire#w1
      Contact( "Blend_T-20".Dose_Sugar.QDOSERun )
   END_RUNG wire#w2
   RUNG wire#w1
      Contact( "Sugar to Mix"."System ready to run" )
      Coil( "Blend_T-20".Dose.Dose_Prod_Ready.%X10 )
   END_RUNG
   RUNG wire#w1
      Contact( "Blend_T-20".Dose_Sugar.QDOSERun )
      Contact( "Sugar to Mix"."Transfer in process" )
      Coil( "General_Blend".Sugar."In Process"."T-20" )
   END_RUNG
   RUNG wire#w1
      Move(in := "Blend to Preparation".Recipe."T-20".Sugar.Sp_DoseQty, out1 => "Blend_T-20".SP_Sugar.Dose_SP)
   END_RUNG
   // the same network as SCL:
   "Blend_T-20".Dose.Dose_Tank_Available.%X10 := "AlwaysTRUE" AND ("Sugar to Mix"."System ready to run" OR "Blend_T-20".Dose_Sugar.QDOSERun);
   "Blend_T-20".Dose.Dose_Prod_Ready.%X10 := "AlwaysTRUE" AND "Sugar to Mix"."System ready to run";
   "General_Blend".Sugar."In Process"."T-20" := "AlwaysTRUE" AND "Blend_T-20".Dose_Sugar.QDOSERun AND "Sugar to Mix"."Transfer in process";
   IF "AlwaysTRUE" THEN
       "Blend_T-20".SP_Sugar.Dose_SP := "Blend to Preparation".Recipe."T-20".Sugar.Sp_DoseQty;
   END_IF;
END_REGION

REGION Network 17: Salt to Blending T-20
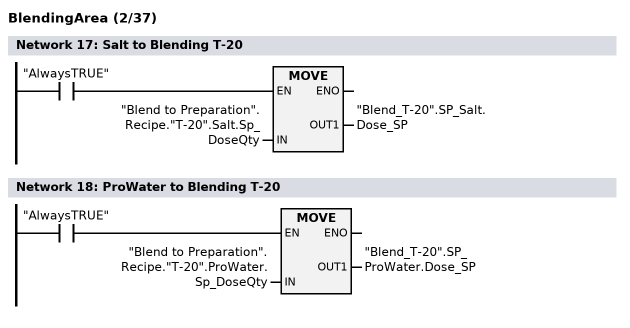
   RUNG wire#powerrail
      Contact( "AlwaysTRUE" )
      Move(in := "Blend to Preparation".Recipe."T-20".Salt.Sp_DoseQty, out1 => "Blend_T-20".SP_Salt.Dose_SP)
   END_RUNG
   // the same network as SCL:
   IF "AlwaysTRUE" THEN
       "Blend_T-20".SP_Salt.Dose_SP := "Blend to Preparation".Recipe."T-20".Salt.Sp_DoseQty;
   END_IF;
END_REGION

REGION Network 18: ProWater to Blending T-20
   RUNG wire#powerrail
      Contact( "AlwaysTRUE" )
      Move(in := "Blend to Preparation".Recipe."T-20".ProWater.Sp_DoseQty, out1 => "Blend_T-20".SP_ProWater.Dose_SP)
   END_RUNG
   // the same network as SCL:
   IF "AlwaysTRUE" THEN
       "Blend_T-20".SP_ProWater.Dose_SP := "Blend to Preparation".Recipe."T-20".ProWater.Sp_DoseQty;
   END_IF;
END_REGION

REGION Network 19: Blending T-20
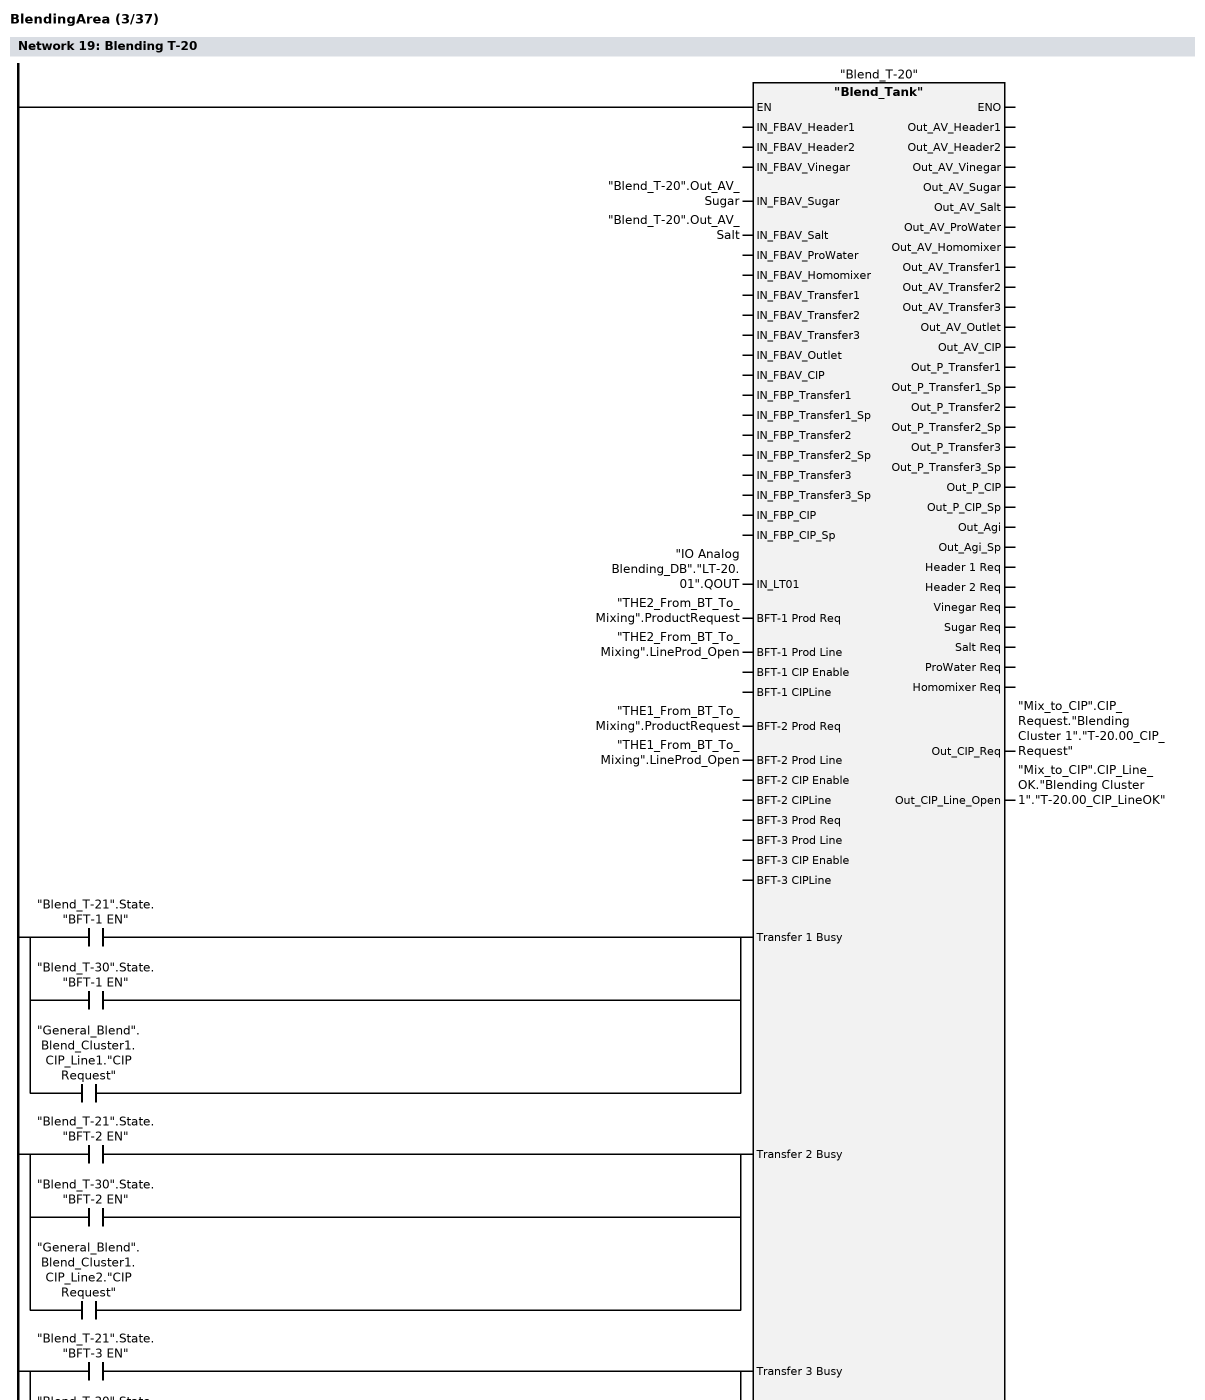
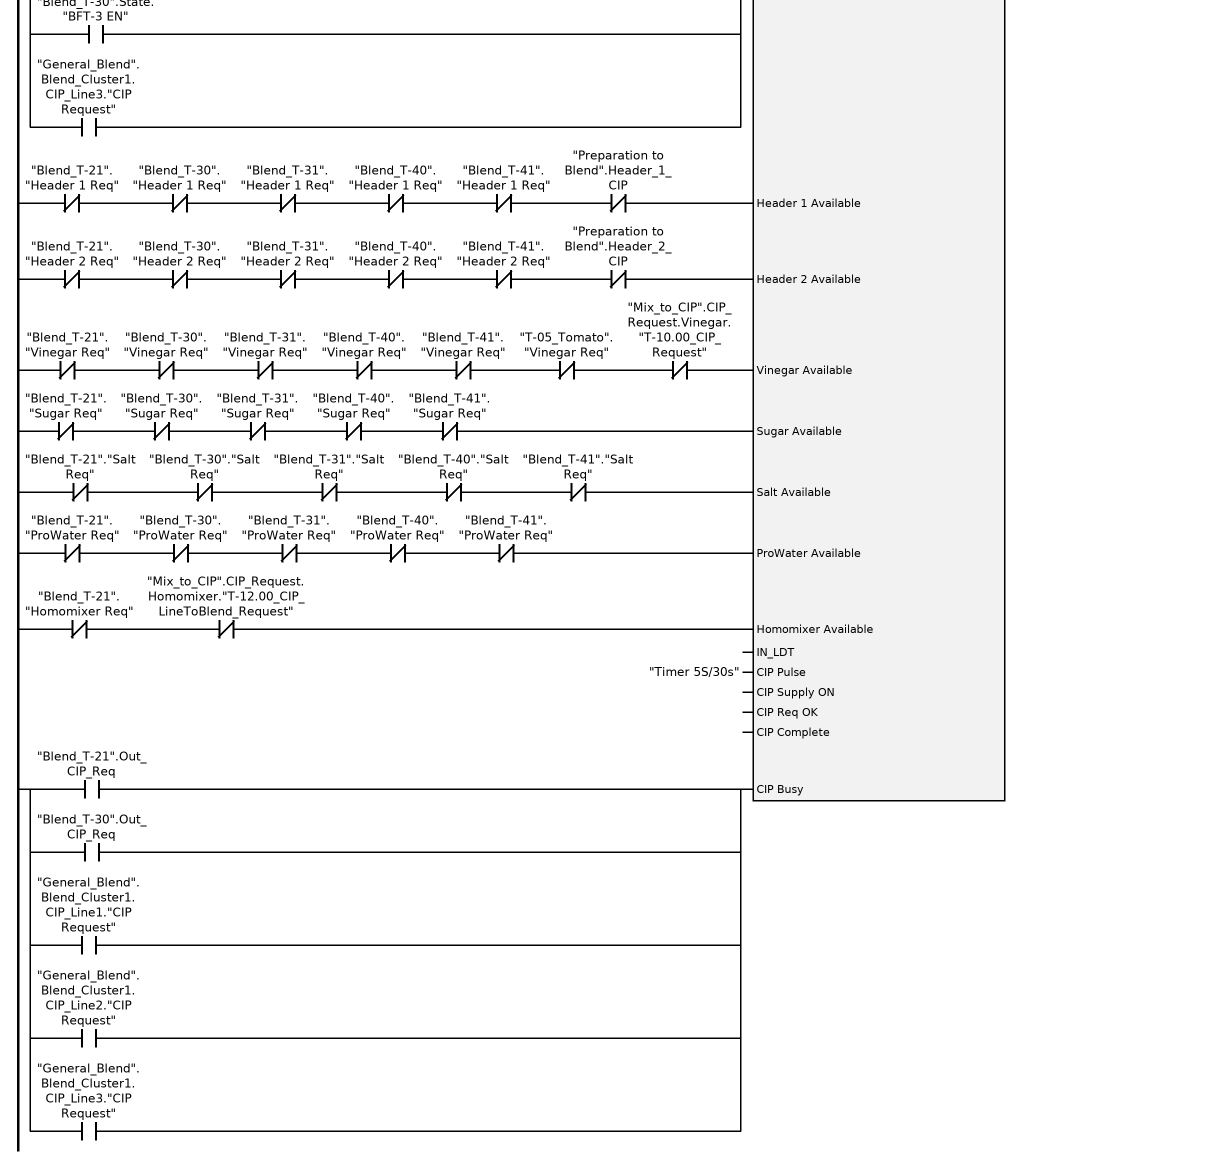
   RUNG wire#powerrail
      "Blend_T-20"("Transfer 1 Busy" := wire#w1, "Transfer 2 Busy" := wire#w2, "Transfer 3 Busy" := wire#w3, "Header 1 Available" := wire#w4, "Header 2 Available" := wire#w5, "Vinegar Available" := wire#w6, "Sugar Available" := wire#w7, "Salt Available" := wire#w8, "ProWater Available" := wire#w9, "Homomixer Available" := wire#w10, "CIP Busy" := wire#w11, IN_FBAV_Header1 :=, IN_FBAV_Header2 :=, IN_FBAV_Vinegar :=, IN_FBAV_Sugar := "Blend_T-20".Out_AV_Sugar, IN_FBAV_Salt := "Blend_T-20".Out_AV_Salt, IN_FBAV_ProWater :=, IN_FBAV_Homomixer :=, IN_FBAV_Transfer1 :=, IN_FBAV_Transfer2 :=, IN_FBAV_Transfer3 :=, IN_FBAV_Outlet :=, IN_FBAV_CIP :=, IN_FBP_Transfer1 :=, IN_FBP_Transfer1_Sp :=, IN_FBP_Transfer2 :=, IN_FBP_Transfer2_Sp :=, IN_FBP_Transfer3 :=, IN_FBP_Transfer3_Sp :=, IN_FBP_CIP :=, IN_FBP_CIP_Sp :=, IN_LT01 := "IO Analog Blending_DB"."LT-20.01".QOUT, "BFT-1 Prod Req" := "THE2_From_BT_To_Mixing".ProductRequest, "BFT-1 Prod Line" := "THE2_From_BT_To_Mixing".LineProd_Open, "BFT-1 CIP Enable" :=, "BFT-1 CIPLine" :=, "BFT-2 Prod Req" := "THE1_From_BT_To_Mixing".ProductRequest, "BFT-2 Prod Line" := "THE1_From_BT_To_Mixing".LineProd_Open, "BFT-2 CIP Enable" :=, "BFT-2 CIPLine" :=, "BFT-3 Prod Req" :=, "BFT-3 Prod Line" :=, "BFT-3 CIP Enable" :=, "BFT-3 CIPLine" :=, IN_LDT :=, "CIP Pulse" := "Timer 5S/30s", "CIP Supply ON" :=, "CIP Req OK" :=, "CIP Complete" :=, Out_AV_Header1 =>, Out_AV_Header2 =>, Out_AV_Vinegar =>, Out_AV_Sugar =>, Out_AV_Salt =>, Out_AV_ProWater =>, Out_AV_Homomixer =>, Out_AV_Transfer1 =>, Out_AV_Transfer2 =>, Out_AV_Transfer3 =>, Out_AV_Outlet =>, Out_AV_CIP =>, Out_P_Transfer1 =>, Out_P_Transfer1_Sp =>, Out_P_Transfer2 =>, Out_P_Transfer2_Sp =>, Out_P_Transfer3 =>, Out_P_Transfer3_Sp =>, Out_P_CIP =>, Out_P_CIP_Sp =>, Out_Agi =>, Out_Agi_Sp =>, "Header 1 Req" =>, "Header 2 Req" =>, "Vinegar Req" =>, "Sugar Req" =>, "Salt Req" =>, "ProWater Req" =>, "Homomixer Req" =>, Out_CIP_Req => "Mix_to_CIP".CIP_Request."Blending Cluster 1"."T-20.00_CIP_Request", Out_CIP_Line_Open => "Mix_to_CIP".CIP_Line_OK."Blending Cluster 1"."T-20.00_CIP_LineOK")
   END_RUNG
   RUNG wire#powerrail
      Contact( "Blend_T-21".State."BFT-1 EN" )
   END_RUNG wire#w1
   RUNG wire#powerrail
      Contact( "Blend_T-30".State."BFT-1 EN" )
   END_RUNG wire#w1
   RUNG wire#powerrail
      Contact( "General_Blend".Blend_Cluster1.CIP_Line1."CIP Request" )
   END_RUNG wire#w1
   RUNG wire#powerrail
      Contact( "Blend_T-21".State."BFT-2 EN" )
   END_RUNG wire#w2
   RUNG wire#powerrail
      Contact( "Blend_T-30".State."BFT-2 EN" )
   END_RUNG wire#w2
   RUNG wire#powerrail
      Contact( "General_Blend".Blend_Cluster1.CIP_Line2."CIP Request" )
   END_RUNG wire#w2
   RUNG wire#powerrail
      Contact( "Blend_T-21".State."BFT-3 EN" )
   END_RUNG wire#w3
   RUNG wire#powerrail
      Contact( "Blend_T-30".State."BFT-3 EN" )
   END_RUNG wire#w3
   RUNG wire#powerrail
      Contact( "General_Blend".Blend_Cluster1.CIP_Line3."CIP Request" )
   END_RUNG wire#w3
   RUNG wire#powerrail
      I_Contact( "Blend_T-21"."Header 1 Req" )
      I_Contact( "Blend_T-30"."Header 1 Req" )
      I_Contact( "Blend_T-31"."Header 1 Req" )
      I_Contact( "Blend_T-40"."Header 1 Req" )
      I_Contact( "Blend_T-41"."Header 1 Req" )
      I_Contact( "Preparation to Blend".Header_1_CIP )
   END_RUNG wire#w4
   RUNG wire#powerrail
      I_Contact( "Blend_T-21"."Header 2 Req" )
      I_Contact( "Blend_T-30"."Header 2 Req" )
      I_Contact( "Blend_T-31"."Header 2 Req" )
      I_Contact( "Blend_T-40"."Header 2 Req" )
      I_Contact( "Blend_T-41"."Header 2 Req" )
      I_Contact( "Preparation to Blend".Header_2_CIP )
   END_RUNG wire#w5
   RUNG wire#powerrail
      I_Contact( "Blend_T-21"."Vinegar Req" )
      I_Contact( "Blend_T-30"."Vinegar Req" )
      I_Contact( "Blend_T-31"."Vinegar Req" )
      I_Contact( "Blend_T-40"."Vinegar Req" )
      I_Contact( "Blend_T-41"."Vinegar Req" )
      I_Contact( "T-05_Tomato"."Vinegar Req" )
      I_Contact( "Mix_to_CIP".CIP_Request.Vinegar."T-10.00_CIP_Request" )
   END_RUNG wire#w6
   RUNG wire#powerrail
      I_Contact( "Blend_T-21"."Sugar Req" )
      I_Contact( "Blend_T-30"."Sugar Req" )
      I_Contact( "Blend_T-31"."Sugar Req" )
      I_Contact( "Blend_T-40"."Sugar Req" )
      I_Contact( "Blend_T-41"."Sugar Req" )
   END_RUNG wire#w7
   RUNG wire#powerrail
      I_Contact( "Blend_T-21"."Salt Req" )
      I_Contact( "Blend_T-30"."Salt Req" )
      I_Contact( "Blend_T-31"."Salt Req" )
      I_Contact( "Blend_T-40"."Salt Req" )
      I_Contact( "Blend_T-41"."Salt Req" )
   END_RUNG wire#w8
   RUNG wire#powerrail
      I_Contact( "Blend_T-21"."ProWater Req" )
      I_Contact( "Blend_T-30"."ProWater Req" )
      I_Contact( "Blend_T-31"."ProWater Req" )
      I_Contact( "Blend_T-40"."ProWater Req" )
      I_Contact( "Blend_T-41"."ProWater Req" )
   END_RUNG wire#w9
   RUNG wire#powerrail
      I_Contact( "Blend_T-21"."Homomixer Req" )
      I_Contact( "Mix_to_CIP".CIP_Request.Homomixer."T-12.00_CIP_LineToBlend_Request" )
   END_RUNG wire#w10
   RUNG wire#powerrail
      Contact( "Blend_T-21".Out_CIP_Req )
   END_RUNG wire#w11
   RUNG wire#powerrail
      Contact( "Blend_T-30".Out_CIP_Req )
   END_RUNG wire#w11
   RUNG wire#powerrail
      Contact( "General_Blend".Blend_Cluster1.CIP_Line1."CIP Request" )
   END_RUNG wire#w11
   RUNG wire#powerrail
      Contact( "General_Blend".Blend_Cluster1.CIP_Line2."CIP Request" )
   END_RUNG wire#w11
   RUNG wire#powerrail
      Contact( "General_Blend".Blend_Cluster1.CIP_Line3."CIP Request" )
   END_RUNG wire#w11
   // the same network as SCL:
   "Blend_T-20"(IN_FBAV_Sugar := "Blend_T-20".Out_AV_Sugar,   // "Blend_Tank"
                IN_FBAV_Salt := "Blend_T-20".Out_AV_Salt,
                IN_LT01 := "IO Analog Blending_DB"."LT-20.01".QOUT,
                "BFT-1 Prod Req" := "THE2_From_BT_To_Mixing".ProductRequest,
                "BFT-1 Prod Line" := "THE2_From_BT_To_Mixing".LineProd_Open,
                "BFT-2 Prod Req" := "THE1_From_BT_To_Mixing".ProductRequest,
                "BFT-2 Prod Line" := "THE1_From_BT_To_Mixing".LineProd_Open,
                "Transfer 1 Busy" := "Blend_T-21".State."BFT-1 EN" OR "Blend_T-30".State."BFT-1 EN" OR "General_Blend".Blend_Cluster1.CIP_Line1."CIP Request",
                "Transfer 2 Busy" := "Blend_T-21".State."BFT-2 EN" OR "Blend_T-30".State."BFT-2 EN" OR "General_Blend".Blend_Cluster1.CIP_Line2."CIP Request",
                "Transfer 3 Busy" := "Blend_T-21".State."BFT-3 EN" OR "Blend_T-30".State."BFT-3 EN" OR "General_Blend".Blend_Cluster1.CIP_Line3."CIP Request",
                "Header 1 Available" := NOT "Blend_T-21"."Header 1 Req" AND NOT "Blend_T-30"."Header 1 Req" AND NOT "Blend_T-31"."Header 1 Req" AND NOT "Blend_T-40"."Header 1 Req" AND NOT "Blend_T-41"."Header 1 Req" AND NOT "Preparation to Blend".Header_1_CIP,
                "Header 2 Available" := NOT "Blend_T-21"."Header 2 Req" AND NOT "Blend_T-30"."Header 2 Req" AND NOT "Blend_T-31"."Header 2 Req" AND NOT "Blend_T-40"."Header 2 Req" AND NOT "Blend_T-41"."Header 2 Req" AND NOT "Preparation to Blend".Header_2_CIP,
                "Vinegar Available" := NOT "Blend_T-21"."Vinegar Req" AND NOT "Blend_T-30"."Vinegar Req" AND NOT "Blend_T-31"."Vinegar Req" AND NOT "Blend_T-40"."Vinegar Req" AND NOT "Blend_T-41"."Vinegar Req" AND NOT "T-05_Tomato"."Vinegar Req" AND NOT "Mix_to_CIP".CIP_Request.Vinegar."T-10.00_CIP_Request",
                "Sugar Available" := NOT "Blend_T-21"."Sugar Req" AND NOT "Blend_T-30"."Sugar Req" AND NOT "Blend_T-31"."Sugar Req" AND NOT "Blend_T-40"."Sugar Req" AND NOT "Blend_T-41"."Sugar Req",
                "Salt Available" := NOT "Blend_T-21"."Salt Req" AND NOT "Blend_T-30"."Salt Req" AND NOT "Blend_T-31"."Salt Req" AND NOT "Blend_T-40"."Salt Req" AND NOT "Blend_T-41"."Salt Req",
                "ProWater Available" := NOT "Blend_T-21"."ProWater Req" AND NOT "Blend_T-30"."ProWater Req" AND NOT "Blend_T-31"."ProWater Req" AND NOT "Blend_T-40"."ProWater Req" AND NOT "Blend_T-41"."ProWater Req",
                "Homomixer Available" := NOT "Blend_T-21"."Homomixer Req" AND NOT "Mix_to_CIP".CIP_Request.Homomixer."T-12.00_CIP_LineToBlend_Request",
                "CIP Pulse" := "Timer 5S/30s",
                "CIP Busy" := "Blend_T-21".Out_CIP_Req OR "Blend_T-30".Out_CIP_Req OR "General_Blend".Blend_Cluster1.CIP_Line1."CIP Request" OR "General_Blend".Blend_Cluster1.CIP_Line2."CIP Request" OR "General_Blend".Blend_Cluster1.CIP_Line3."CIP Request",
                Out_CIP_Req => "Mix_to_CIP".CIP_Request."Blending Cluster 1"."T-20.00_CIP_Request",
                Out_CIP_Line_Open => "Mix_to_CIP".CIP_Line_OK."Blending Cluster 1"."T-20.00_CIP_LineOK");
END_REGION

REGION Network 20: Blending T-20 Feedback Valve
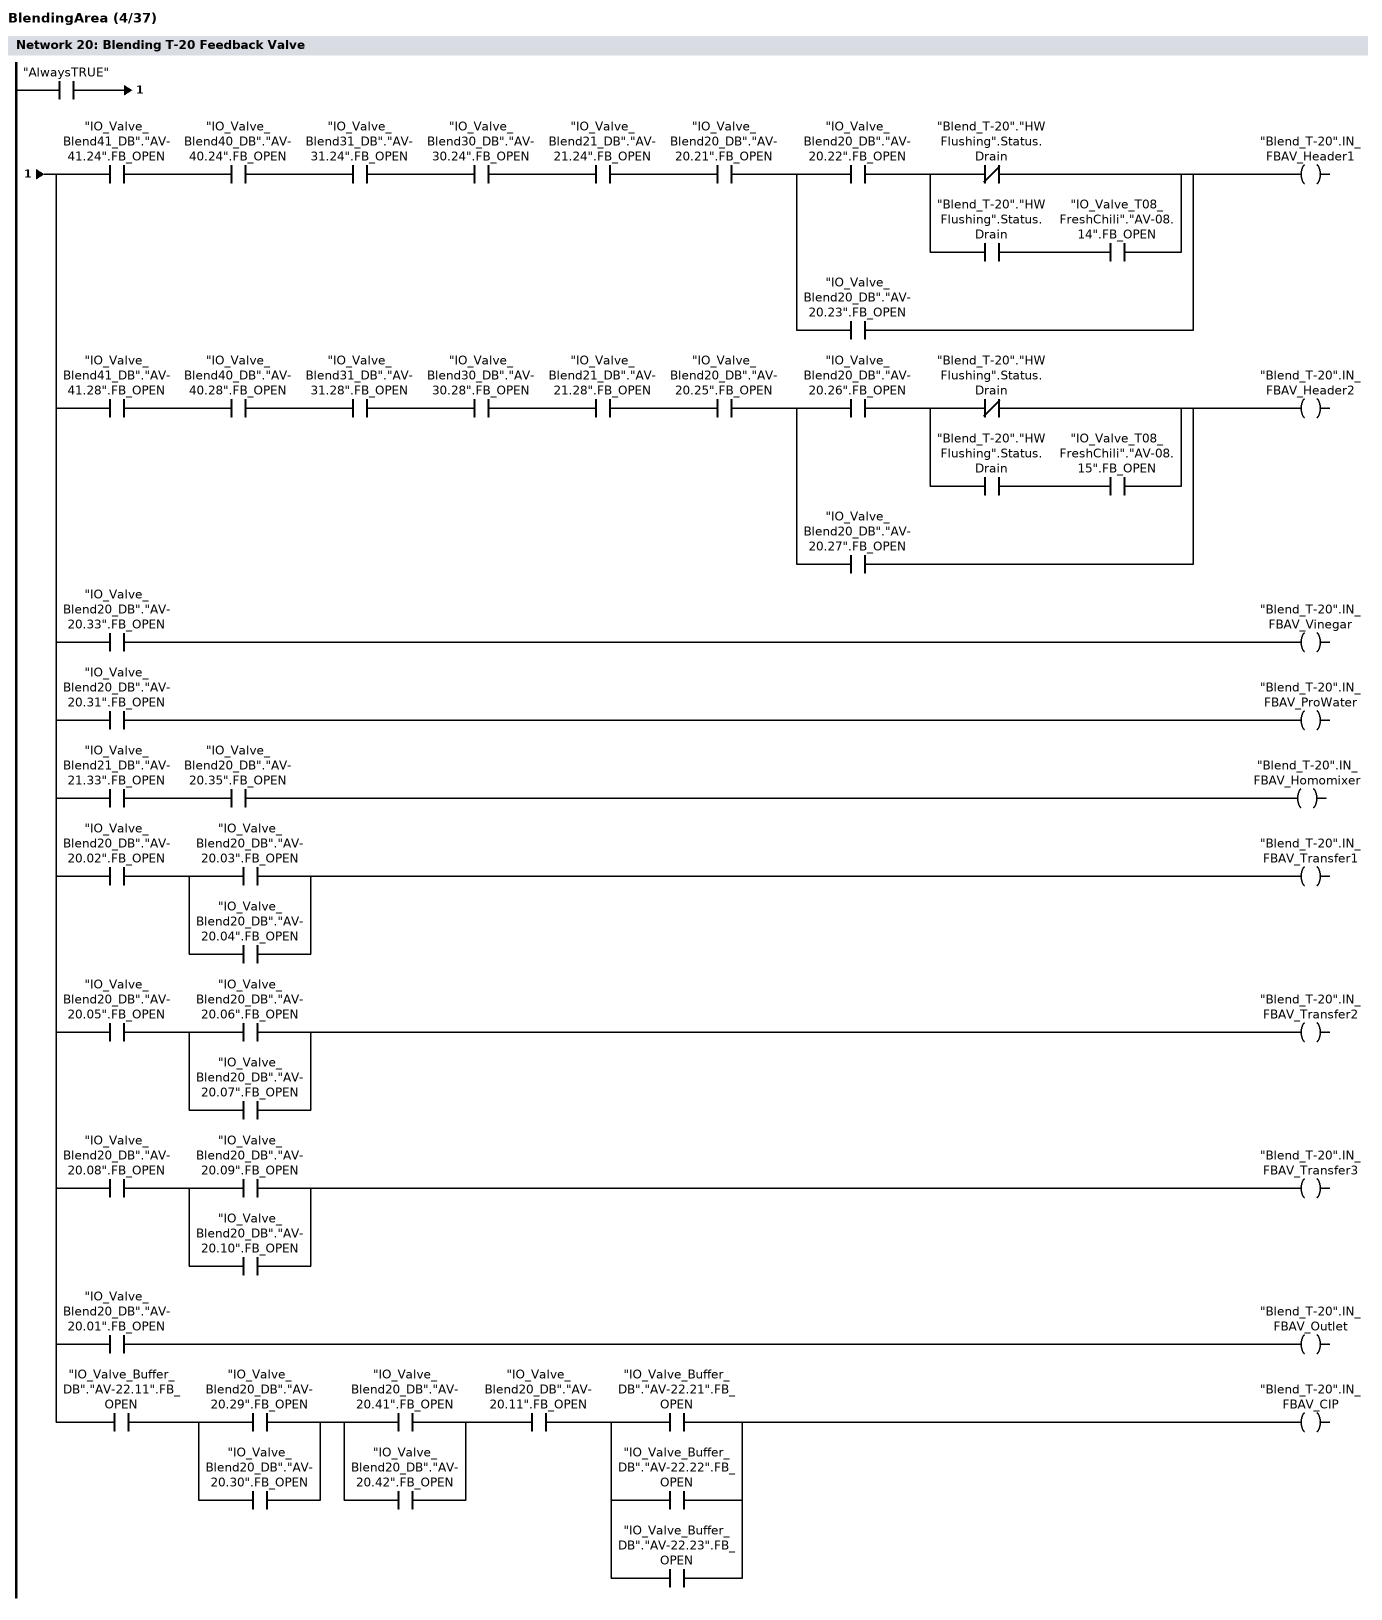
   RUNG wire#powerrail
      Contact( "AlwaysTRUE" )
      wire#w1
      Contact( "IO_Valve_Blend41_DB"."AV-41.24".FB_OPEN )
      Contact( "IO_Valve_Blend40_DB"."AV-40.24".FB_OPEN )
      Contact( "IO_Valve_Blend31_DB"."AV-31.24".FB_OPEN )
      Contact( "IO_Valve_Blend30_DB"."AV-30.24".FB_OPEN )
      Contact( "IO_Valve_Blend21_DB"."AV-21.24".FB_OPEN )
      Contact( "IO_Valve_Blend20_DB"."AV-20.21".FB_OPEN )
      wire#w2
      Contact( "IO_Valve_Blend20_DB"."AV-20.22".FB_OPEN )
      wire#w3
      I_Contact( "Blend_T-20"."HW Flushing".Status.Drain )
      wire#w4
      Coil( "Blend_T-20".IN_FBAV_Header1 )
   END_RUNG
   RUNG wire#w3
      Contact( "Blend_T-20"."HW Flushing".Status.Drain )
      Contact( "IO_Valve_T08_FreshChili"."AV-08.14".FB_OPEN )
   END_RUNG wire#w4
   RUNG wire#w2
      Contact( "IO_Valve_Blend20_DB"."AV-20.23".FB_OPEN )
   END_RUNG wire#w4
   RUNG wire#w1
      Contact( "IO_Valve_Blend41_DB"."AV-41.28".FB_OPEN )
      Contact( "IO_Valve_Blend40_DB"."AV-40.28".FB_OPEN )
      Contact( "IO_Valve_Blend31_DB"."AV-31.28".FB_OPEN )
      Contact( "IO_Valve_Blend30_DB"."AV-30.28".FB_OPEN )
      Contact( "IO_Valve_Blend21_DB"."AV-21.28".FB_OPEN )
      Contact( "IO_Valve_Blend20_DB"."AV-20.25".FB_OPEN )
      wire#w5
      Contact( "IO_Valve_Blend20_DB"."AV-20.26".FB_OPEN )
      wire#w6
      I_Contact( "Blend_T-20"."HW Flushing".Status.Drain )
      wire#w7
      Coil( "Blend_T-20".IN_FBAV_Header2 )
   END_RUNG
   RUNG wire#w6
      Contact( "Blend_T-20"."HW Flushing".Status.Drain )
      Contact( "IO_Valve_T08_FreshChili"."AV-08.15".FB_OPEN )
   END_RUNG wire#w7
   RUNG wire#w5
      Contact( "IO_Valve_Blend20_DB"."AV-20.27".FB_OPEN )
   END_RUNG wire#w7
   RUNG wire#w1
      Contact( "IO_Valve_Blend20_DB"."AV-20.33".FB_OPEN )
      Coil( "Blend_T-20".IN_FBAV_Vinegar )
   END_RUNG
   RUNG wire#w1
      Contact( "IO_Valve_Blend20_DB"."AV-20.31".FB_OPEN )
      Coil( "Blend_T-20".IN_FBAV_ProWater )
   END_RUNG
   RUNG wire#w1
      Contact( "IO_Valve_Blend21_DB"."AV-21.33".FB_OPEN )
      Contact( "IO_Valve_Blend20_DB"."AV-20.35".FB_OPEN )
      Coil( "Blend_T-20".IN_FBAV_Homomixer )
   END_RUNG
   RUNG wire#w1
      Contact( "IO_Valve_Blend20_DB"."AV-20.02".FB_OPEN )
      wire#w8
      Contact( "IO_Valve_Blend20_DB"."AV-20.03".FB_OPEN )
      wire#w9
      Coil( "Blend_T-20".IN_FBAV_Transfer1 )
   END_RUNG
   RUNG wire#w8
      Contact( "IO_Valve_Blend20_DB"."AV-20.04".FB_OPEN )
   END_RUNG wire#w9
   RUNG wire#w1
      Contact( "IO_Valve_Blend20_DB"."AV-20.05".FB_OPEN )
      wire#w10
      Contact( "IO_Valve_Blend20_DB"."AV-20.06".FB_OPEN )
      wire#w11
      Coil( "Blend_T-20".IN_FBAV_Transfer2 )
   END_RUNG
   RUNG wire#w10
      Contact( "IO_Valve_Blend20_DB"."AV-20.07".FB_OPEN )
   END_RUNG wire#w11
   RUNG wire#w1
      Contact( "IO_Valve_Blend20_DB"."AV-20.08".FB_OPEN )
      wire#w12
      Contact( "IO_Valve_Blend20_DB"."AV-20.09".FB_OPEN )
      wire#w13
      Coil( "Blend_T-20".IN_FBAV_Transfer3 )
   END_RUNG
   RUNG wire#w12
      Contact( "IO_Valve_Blend20_DB"."AV-20.10".FB_OPEN )
   END_RUNG wire#w13
   RUNG wire#w1
      Contact( "IO_Valve_Blend20_DB"."AV-20.01".FB_OPEN )
      Coil( "Blend_T-20".IN_FBAV_Outlet )
   END_RUNG
   RUNG wire#w1
      Contact( "IO_Valve_Buffer_DB"."AV-22.11".FB_OPEN )
      wire#w14
      Contact( "IO_Valve_Blend20_DB"."AV-20.29".FB_OPEN )
      wire#w15
      Contact( "IO_Valve_Blend20_DB"."AV-20.41".FB_OPEN )
      wire#w16
      Contact( "IO_Valve_Blend20_DB"."AV-20.11".FB_OPEN )
      wire#w17
      Contact( "IO_Valve_Buffer_DB"."AV-22.21".FB_OPEN )
      wire#w18
      Coil( "Blend_T-20".IN_FBAV_CIP )
   END_RUNG
   RUNG wire#w14
      Contact( "IO_Valve_Blend20_DB"."AV-20.30".FB_OPEN )
   END_RUNG wire#w15
   RUNG wire#w15
      Contact( "IO_Valve_Blend20_DB"."AV-20.42".FB_OPEN )
   END_RUNG wire#w16
   RUNG wire#w17
      Contact( "IO_Valve_Buffer_DB"."AV-22.22".FB_OPEN )
   END_RUNG wire#w18
   RUNG wire#w17
      Contact( "IO_Valve_Buffer_DB"."AV-22.23".FB_OPEN )
   END_RUNG wire#w18
   // the same network as SCL:
   "Blend_T-20".IN_FBAV_Header1 := "AlwaysTRUE" AND "IO_Valve_Blend41_DB"."AV-41.24".FB_OPEN AND "IO_Valve_Blend40_DB"."AV-40.24".FB_OPEN AND "IO_Valve_Blend31_DB"."AV-31.24".FB_OPEN AND "IO_Valve_Blend30_DB"."AV-30.24".FB_OPEN AND "IO_Valve_Blend21_DB"."AV-21.24".FB_OPEN AND "IO_Valve_Blend20_DB"."AV-20.21".FB_OPEN AND (("IO_Valve_Blend20_DB"."AV-20.22".FB_OPEN AND (NOT "Blend_T-20"."HW Flushing".Status.Drain OR ("Blend_T-20"."HW Flushing".Status.Drain AND "IO_Valve_T08_FreshChili"."AV-08.14".FB_OPEN))) OR "IO_Valve_Blend20_DB"."AV-20.23".FB_OPEN);
   "Blend_T-20".IN_FBAV_Header2 := "AlwaysTRUE" AND "IO_Valve_Blend41_DB"."AV-41.28".FB_OPEN AND "IO_Valve_Blend40_DB"."AV-40.28".FB_OPEN AND "IO_Valve_Blend31_DB"."AV-31.28".FB_OPEN AND "IO_Valve_Blend30_DB"."AV-30.28".FB_OPEN AND "IO_Valve_Blend21_DB"."AV-21.28".FB_OPEN AND "IO_Valve_Blend20_DB"."AV-20.25".FB_OPEN AND (("IO_Valve_Blend20_DB"."AV-20.26".FB_OPEN AND (NOT "Blend_T-20"."HW Flushing".Status.Drain OR ("Blend_T-20"."HW Flushing".Status.Drain AND "IO_Valve_T08_FreshChili"."AV-08.15".FB_OPEN))) OR "IO_Valve_Blend20_DB"."AV-20.27".FB_OPEN);
   "Blend_T-20".IN_FBAV_Vinegar := "AlwaysTRUE" AND "IO_Valve_Blend20_DB"."AV-20.33".FB_OPEN;
   "Blend_T-20".IN_FBAV_ProWater := "AlwaysTRUE" AND "IO_Valve_Blend20_DB"."AV-20.31".FB_OPEN;
   "Blend_T-20".IN_FBAV_Homomixer := "AlwaysTRUE" AND "IO_Valve_Blend21_DB"."AV-21.33".FB_OPEN AND "IO_Valve_Blend20_DB"."AV-20.35".FB_OPEN;
   "Blend_T-20".IN_FBAV_Transfer1 := "AlwaysTRUE" AND "IO_Valve_Blend20_DB"."AV-20.02".FB_OPEN AND ("IO_Valve_Blend20_DB"."AV-20.03".FB_OPEN OR "IO_Valve_Blend20_DB"."AV-20.04".FB_OPEN);
   "Blend_T-20".IN_FBAV_Transfer2 := "AlwaysTRUE" AND "IO_Valve_Blend20_DB"."AV-20.05".FB_OPEN AND ("IO_Valve_Blend20_DB"."AV-20.06".FB_OPEN OR "IO_Valve_Blend20_DB"."AV-20.07".FB_OPEN);
   "Blend_T-20".IN_FBAV_Transfer3 := "AlwaysTRUE" AND "IO_Valve_Blend20_DB"."AV-20.08".FB_OPEN AND ("IO_Valve_Blend20_DB"."AV-20.09".FB_OPEN OR "IO_Valve_Blend20_DB"."AV-20.10".FB_OPEN);
   "Blend_T-20".IN_FBAV_Outlet := "AlwaysTRUE" AND "IO_Valve_Blend20_DB"."AV-20.01".FB_OPEN;
   "Blend_T-20".IN_FBAV_CIP := "AlwaysTRUE" AND "IO_Valve_Buffer_DB"."AV-22.11".FB_OPEN AND ("IO_Valve_Blend20_DB"."AV-20.29".FB_OPEN OR "IO_Valve_Blend20_DB"."AV-20.30".FB_OPEN) AND ("IO_Valve_Blend20_DB"."AV-20.41".FB_OPEN OR "IO_Valve_Blend20_DB"."AV-20.42".FB_OPEN) AND "IO_Valve_Blend20_DB"."AV-20.11".FB_OPEN AND ("IO_Valve_Buffer_DB"."AV-22.21".FB_OPEN OR "IO_Valve_Buffer_DB"."AV-22.22".FB_OPEN OR "IO_Valve_Buffer_DB"."AV-22.23".FB_OPEN);
END_REGION

REGION Network 21: Blending T-20 Feedback Pump
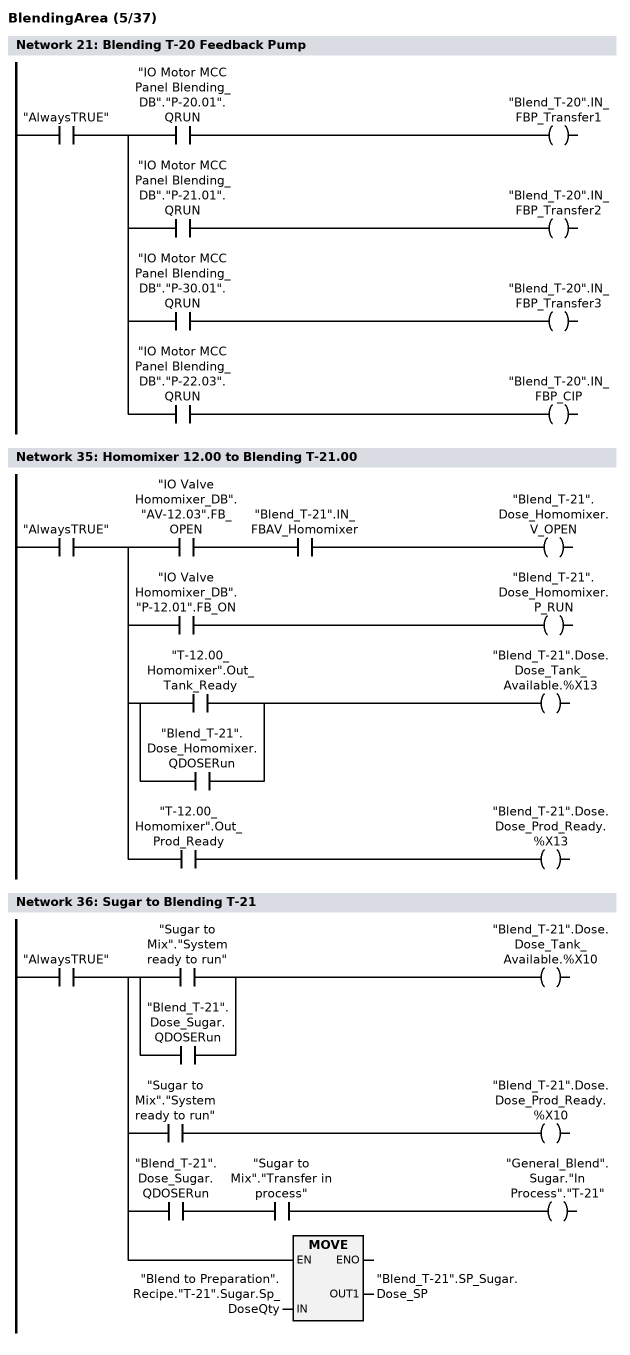
   RUNG wire#powerrail
      Contact( "AlwaysTRUE" )
      wire#w1
      Contact( "IO Motor MCC Panel Blending_DB"."P-20.01".QRUN )
      Coil( "Blend_T-20".IN_FBP_Transfer1 )
   END_RUNG
   RUNG wire#w1
      Contact( "IO Motor MCC Panel Blending_DB"."P-21.01".QRUN )
      Coil( "Blend_T-20".IN_FBP_Transfer2 )
   END_RUNG
   RUNG wire#w1
      Contact( "IO Motor MCC Panel Blending_DB"."P-30.01".QRUN )
      Coil( "Blend_T-20".IN_FBP_Transfer3 )
   END_RUNG
   RUNG wire#w1
      Contact( "IO Motor MCC Panel Blending_DB"."P-22.03".QRUN )
      Coil( "Blend_T-20".IN_FBP_CIP )
   END_RUNG
   // the same network as SCL:
   "Blend_T-20".IN_FBP_Transfer1 := "AlwaysTRUE" AND "IO Motor MCC Panel Blending_DB"."P-20.01".QRUN;
   "Blend_T-20".IN_FBP_Transfer2 := "AlwaysTRUE" AND "IO Motor MCC Panel Blending_DB"."P-21.01".QRUN;
   "Blend_T-20".IN_FBP_Transfer3 := "AlwaysTRUE" AND "IO Motor MCC Panel Blending_DB"."P-30.01".QRUN;
   "Blend_T-20".IN_FBP_CIP := "AlwaysTRUE" AND "IO Motor MCC Panel Blending_DB"."P-22.03".QRUN;
END_REGION

NETWORK
TITLE = Blending T-20 to Preparation
//to ChiliAwetan1
      O     "Blend_T-20".Dose_ChiliAwetan1.QDOSERun;  //Dose Run
      =     "Blend to Preparation"."T-20".Raw_Material.ChiliAwetan_1.DoseRun;
      O     "Blend_T-20".Dose_ChiliAwetan1.QHELD;  //Dose Held
      =     "Blend to Preparation"."T-20".Raw_Material.ChiliAwetan_1.DoseHeld;
      O     "Blend_T-20".Dose_ChiliAwetan1.QDoseComplete;  //Dose Complete
      =     "Blend to Preparation"."T-20".Raw_Material.ChiliAwetan_1.DoseComplete;
      O     "Blend_T-20".Dose_ChiliAwetan1.V_CMD;  //Valve Command
      =     "Blend to Preparation"."T-20".Raw_Material.ChiliAwetan_1.ValveCMD;
      O     "Blend_T-20".Dose_ChiliAwetan1.P_CMD;  //Pump Command
      =     "Blend to Preparation"."T-20".Raw_Material.ChiliAwetan_1.PumpCMD;
      O     "Blend_T-20".Dose.Dose_Header_Req.%X0;  //Header 1 Req
      =     "Blend to Preparation"."T-20".Raw_Material.ChiliAwetan_1.Header1_Req;
      O     "Blend_T-20".Dose.Dose_Header_Req.%X16;  //Header 2 Req
      =     "Blend to Preparation"."T-20".Raw_Material.ChiliAwetan_1.Header2_Req;
      L     "Blend to Preparation".Recipe."T-20".ChiliAwetan_1.Sp_DoseQty;  //Load Sp Dose From Recipe
      T     "Blend_T-20".SP_ChiliAwetan1.Dose_SP;
      L     "Blend_T-20".Dose_ChiliAwetan1.P_SPEED;  //Pump Speed
      T     "Blend to Preparation".Recipe."T-20".ChiliAwetan_1.SP_PumpSpeed;

//to ChiliAwetan2
      O     "Blend_T-20".Dose_ChiliAwetan2.QDOSERun;  //Dose Run
      =     "Blend to Preparation"."T-20".Raw_Material.ChiliAwetan_2.DoseRun;
      O     "Blend_T-20".Dose_ChiliAwetan2.QHELD;  //Dose Held
      =     "Blend to Preparation"."T-20".Raw_Material.ChiliAwetan_2.DoseHeld;
      O     "Blend_T-20".Dose_ChiliAwetan2.QDoseComplete;  //Dose Complete
      =     "Blend to Preparation"."T-20".Raw_Material.ChiliAwetan_2.DoseComplete;
      O     "Blend_T-20".Dose_ChiliAwetan2.V_CMD;  //Valve Command
      =     "Blend to Preparation"."T-20".Raw_Material.ChiliAwetan_2.ValveCMD;
      O     "Blend_T-20".Dose_ChiliAwetan2.P_CMD;  //Pump Command
      =     "Blend to Preparation"."T-20".Raw_Material.ChiliAwetan_2.PumpCMD;
      O     "Blend_T-20".Dose.Dose_Header_Req.%X1;  //Header 1 Req
      =     "Blend to Preparation"."T-20".Raw_Material.ChiliAwetan_2.Header1_Req;
      O     "Blend_T-20".Dose.Dose_Header_Req.%X17;  //Header 2 Req
      =     "Blend to Preparation"."T-20".Raw_Material.ChiliAwetan_2.Header2_Req;
      L     "Blend to Preparation".Recipe."T-20".ChiliAwetan_2.Sp_DoseQty;  //Load Sp Dose From Recipe
      T     "Blend_T-20".SP_ChiliAwetan2.Dose_SP;
      L     "Blend_T-20".Dose_ChiliAwetan2.P_SPEED;  //Pump Speed
      T     "Blend to Preparation".Recipe."T-20".ChiliAwetan_2.SP_PumpSpeed;

//to ChiliAwetan3
      O     "Blend_T-20".Dose_ChiliAwetan3.QDOSERun;  //Dose Run
      =     "Blend to Preparation"."T-20".Raw_Material.ChiliAwetan_3.DoseRun;
      O     "Blend_T-20".Dose_ChiliAwetan3.QHELD;  //Dose Held
      =     "Blend to Preparation"."T-20".Raw_Material.ChiliAwetan_3.DoseHeld;
      O     "Blend_T-20".Dose_ChiliAwetan3.QDoseComplete;  //Dose Complete
      =     "Blend to Preparation"."T-20".Raw_Material.ChiliAwetan_3.DoseComplete;
      O     "Blend_T-20".Dose_ChiliAwetan3.V_CMD;  //Valve Command
      =     "Blend to Preparation"."T-20".Raw_Material.ChiliAwetan_3.ValveCMD;
      O     "Blend_T-20".Dose_ChiliAwetan3.P_CMD;  //Pump Command
      =     "Blend to Preparation"."T-20".Raw_Material.ChiliAwetan_3.PumpCMD;
      O     "Blend_T-20".Dose.Dose_Header_Req.%X2;  //Header 1 Req
      =     "Blend to Preparation"."T-20".Raw_Material.ChiliAwetan_3.Header1_Req;
      O     "Blend_T-20".Dose.Dose_Header_Req.%X18;  //Header 2 Req
      =     "Blend to Preparation"."T-20".Raw_Material.ChiliAwetan_3.Header2_Req;
      L     "Blend to Preparation".Recipe."T-20".ChiliAwetan_3.Sp_DoseQty;  //Load Sp Dose From Recipe
      T     "Blend_T-20".SP_ChiliAwetan3.Dose_SP;
      L     "Blend_T-20".Dose_ChiliAwetan3.P_SPEED;  //Pump Speed
      T     "Blend to Preparation".Recipe."T-20".ChiliAwetan_3.SP_PumpSpeed;

//to Tomato
      O     "Blend_T-20".Dose_Tomato.QDOSERun;  //Dose Run
      =     "Blend to Preparation"."T-20".Raw_Material.Tomato.DoseRun;
      O     "Blend_T-20".Dose_Tomato.QHELD;  //Dose Held
      =     "Blend to Preparation"."T-20".Raw_Material.Tomato.DoseHeld;
      O     "Blend_T-20".Dose_Tomato.QDoseComplete;  //Dose Complete
      =     "Blend to Preparation"."T-20".Raw_Material.Tomato.DoseComplete;
      O     "Blend_T-20".Dose_Tomato.V_CMD;  //Valve Command
      =     "Blend to Preparation"."T-20".Raw_Material.Tomato.ValveCMD;
      O     "Blend_T-20".Dose_Tomato.P_CMD;  //Pump Command
      =     "Blend to Preparation"."T-20".Raw_Material.Tomato.PumpCMD;
      O     "Blend_T-20".Dose.Dose_Header_Req.%X3;  //Header 1 Req
      =     "Blend to Preparation"."T-20".Raw_Material.Tomato.Header1_Req;
      O     "Blend_T-20".Dose.Dose_Header_Req.%X19;  //Header 2 Req
      =     "Blend to Preparation"."T-20".Raw_Material.Tomato.Header2_Req;
      L     "Blend to Preparation".Recipe."T-20".Tomato.Sp_DoseQty;  //Load Sp Dose From Recipe
      T     "Blend_T-20".SP_Tomato.Dose_SP;
      L     "Blend_T-20".Dose_Tomato.P_SPEED;  //Pump Speed
      T     "Blend to Preparation".Recipe."T-20".Tomato.SP_PumpSpeed;

//to ChiliFresh1
      O     "Blend_T-20".Dose_ChiliFresh1.QDOSERun;  //Dose Run
      =     "Blend to Preparation"."T-20".Raw_Material.ChiliFresh_1.DoseRun;
      O     "Blend_T-20".Dose_ChiliFresh1.QHELD;  //Dose Held
      =     "Blend to Preparation"."T-20".Raw_Material.ChiliFresh_1.DoseHeld;
      O     "Blend_T-20".Dose_ChiliFresh1.QDoseComplete;  //Dose Complete
      =     "Blend to Preparation"."T-20".Raw_Material.ChiliFresh_1.DoseComplete;
      O     "Blend_T-20".Dose_ChiliFresh1.V_CMD;  //Valve Command
      =     "Blend to Preparation"."T-20".Raw_Material.ChiliFresh_1.ValveCMD;
      O     "Blend_T-20".Dose_ChiliFresh1.P_CMD;  //Pump Command
      =     "Blend to Preparation"."T-20".Raw_Material.ChiliFresh_1.PumpCMD;
      O     "Blend_T-20".Dose.Dose_Header_Req.%X4;  //Header 1 Req
      =     "Blend to Preparation"."T-20".Raw_Material.ChiliFresh_1.Header1_Req;
      O     "Blend_T-20".Dose.Dose_Header_Req.%X20;  //Header 2 Req
      =     "Blend to Preparation"."T-20".Raw_Material.ChiliFresh_1.Header2_Req;
      L     "Blend to Preparation".Recipe."T-20".ChiliFresh_1.Sp_DoseQty;  //Load Sp Dose From Recipe
      T     "Blend_T-20".SP_ChiliFresh1.Dose_SP;
      L     "Blend_T-20".Dose_ChiliFresh1.P_SPEED;  //Pump Speed
      T     "Blend to Preparation".Recipe."T-20".ChiliFresh_1.SP_PumpSpeed;

//to ChiliFresh2
      O     "Blend_T-20".Dose_ChiliFresh2.QDOSERun;  //Dose Run
      =     "Blend to Preparation"."T-20".Raw_Material.ChiliFresh_2.DoseRun;
      O     "Blend_T-20".Dose_ChiliFresh2.QHELD;  //Dose Held
      =     "Blend to Preparation"."T-20".Raw_Material.ChiliFresh_2.DoseHeld;
      O     "Blend_T-20".Dose_ChiliFresh2.QDoseComplete;  //Dose Complete
      =     "Blend to Preparation"."T-20".Raw_Material.ChiliFresh_2.DoseComplete;
      O     "Blend_T-20".Dose_ChiliFresh2.V_CMD;  //Valve Command
      =     "Blend to Preparation"."T-20".Raw_Material.ChiliFresh_2.ValveCMD;
      O     "Blend_T-20".Dose_ChiliFresh2.P_CMD;  //Pump Command
      =     "Blend to Preparation"."T-20".Raw_Material.ChiliFresh_2.PumpCMD;
      O     "Blend_T-20".Dose.Dose_Header_Req.%X5;  //Header 1 Req
      =     "Blend to Preparation"."T-20".Raw_Material.ChiliFresh_2.Header1_Req;
      O     "Blend_T-20".Dose.Dose_Header_Req.%X21;  //Header 2 Req
      =     "Blend to Preparation"."T-20".Raw_Material.ChiliFresh_2.Header2_Req;
      L     "Blend to Preparation".Recipe."T-20".ChiliFresh_2.Sp_DoseQty;  //Load Sp Dose From Recipe
      T     "Blend_T-20".SP_ChiliFresh2.Dose_SP;
      L     "Blend_T-20".Dose_ChiliFresh2.P_SPEED;  //Pump Speed
      T     "Blend to Preparation".Recipe."T-20".ChiliFresh_2.SP_PumpSpeed;

//to ChiliFresh3
      O     "Blend_T-20".Dose_ChiliFresh3.QDOSERun;  //Dose Run
      =     "Blend to Preparation"."T-20".Raw_Material.ChiliFresh_3.DoseRun;
      O     "Blend_T-20".Dose_ChiliFresh3.QHELD;  //Dose Held
      =     "Blend to Preparation"."T-20".Raw_Material.ChiliFresh_3.DoseHeld;
      O     "Blend_T-20".Dose_ChiliFresh3.QDoseComplete;  //Dose Complete
      =     "Blend to Preparation"."T-20".Raw_Material.ChiliFresh_3.DoseComplete;
      O     "Blend_T-20".Dose_ChiliFresh3.V_CMD;  //Valve Command
      =     "Blend to Preparation"."T-20".Raw_Material.ChiliFresh_3.ValveCMD;
      O     "Blend_T-20".Dose_ChiliFresh3.P_CMD;  //Pump Command
      =     "Blend to Preparation"."T-20".Raw_Material.ChiliFresh_3.PumpCMD;
      O     "Blend_T-20".Dose.Dose_Header_Req.%X6;  //Header 1 Req
      =     "Blend to Preparation"."T-20".Raw_Material.ChiliFresh_3.Header1_Req;
      O     "Blend_T-20".Dose.Dose_Header_Req.%X22;  //Header 2 Req
      =     "Blend to Preparation"."T-20".Raw_Material.ChiliFresh_3.Header2_Req;
      L     "Blend to Preparation".Recipe."T-20".ChiliFresh_3.Sp_DoseQty;  //Load Sp Dose From Recipe
      T     "Blend_T-20".SP_ChiliFresh3.Dose_SP;
      L     "Blend_T-20".Dose_ChiliFresh3.P_SPEED;  //Pump Speed
      T     "Blend to Preparation".Recipe."T-20".ChiliFresh_3.SP_PumpSpeed;

//to Garlic
      O     "Blend_T-20".Dose_Garlic.QDOSERun;  //Dose Run
      =     "Blend to Preparation"."T-20".Raw_Material.Garlic.DoseRun;
      O     "Blend_T-20".Dose_Garlic.QHELD;  //Dose Held
      =     "Blend to Preparation"."T-20".Raw_Material.Garlic.DoseHeld;
      O     "Blend_T-20".Dose_Garlic.QDoseComplete;  //Dose Complete
      =     "Blend to Preparation"."T-20".Raw_Material.Garlic.DoseComplete;
      O     "Blend_T-20".Dose_Garlic.V_CMD;  //Valve Command
      =     "Blend to Preparation"."T-20".Raw_Material.Garlic.ValveCMD;
      O     "Blend_T-20".Dose_Garlic.P_CMD;  //Pump Command
      =     "Blend to Preparation"."T-20".Raw_Material.Garlic.PumpCMD;
      O     "Blend_T-20".Dose.Dose_Header_Req.%X7;  //Header 1 Req
      =     "Blend to Preparation"."T-20".Raw_Material.Garlic.Header1_Req;
      O     "Blend_T-20".Dose.Dose_Header_Req.%X23;  //Header 2 Req
      =     "Blend to Preparation"."T-20".Raw_Material.Garlic.Header2_Req;
      L     "Blend to Preparation".Recipe."T-20".Garlic.Sp_DoseQty;  //Load Sp Dose From Recipe
      T     "Blend_T-20".SP_Garlic.Dose_SP;
      L     "Blend_T-20".Dose_Garlic.P_SPEED;  //Pump Speed
      T     "Blend to Preparation".Recipe."T-20".Garlic.SP_PumpSpeed;

//to Vinegar
      O     "Blend_T-20".Dose_Vinegar.QDOSERun;  //Dose Run
      =     "Blend to Preparation"."T-20".Raw_Material.Vinegar.DoseRun;
      O     "Blend_T-20".Dose_Vinegar.QHELD;  //Dose Held
      =     "Blend to Preparation"."T-20".Raw_Material.Vinegar.DoseHeld;
      O     "Blend_T-20".Dose_Vinegar.QDoseComplete;  //Dose Complete
      =     "Blend to Preparation"."T-20".Raw_Material.Vinegar.DoseComplete;
      O     "Blend_T-20".Dose_Vinegar.V_CMD;  //Valve Command
      =     "Blend to Preparation"."T-20".Raw_Material.Vinegar.ValveCMD;
      O     "Blend_T-20".Dose_Vinegar.P_CMD;  //Pump Command
      =     "Blend to Preparation"."T-20".Raw_Material.Vinegar.PumpCMD;
      L     "Blend to Preparation".Recipe."T-20".Vinegar.Sp_DoseQty;  //Load Sp Dose From Recipe
      T     "Blend_T-20".SP_Vinegar.Dose_SP;
      L     "Blend_T-20".Dose_Vinegar.P_SPEED;  //Pump Speed
      T     "Blend to Preparation".Recipe."T-20".Vinegar.SP_PumpSpeed;

//to HW
      O     "Blend_T-20".Dose_HW.QDOSERun;  //Dose Run
      =     "Blend to Preparation"."T-20".Raw_Material.HW.DoseRun;
      O     "Blend_T-20".Dose_HW.QHELD;  //Dose Held
      =     "Blend to Preparation"."T-20".Raw_Material.HW.DoseHeld;
      O     "Blend_T-20".Dose_HW.QDoseComplete;  //Dose Complete
      =     "Blend to Preparation"."T-20".Raw_Material.HW.DoseComplete;
      O     "Blend_T-20".Dose_HW.V_CMD;  //Valve Command
      =     "Blend to Preparation"."T-20".Raw_Material.HW.ValveCMD;
      O     "Blend_T-20".Dose_HW.P_CMD;  //Pump Command
      =     "Blend to Preparation"."T-20".Raw_Material.HW.PumpCMD;
      O     "Blend_T-20".Dose.Dose_Header_Req.%X8;  //Header 1 Req
      =     "Blend to Preparation"."T-20".Raw_Material.HW.Header1_Req;
      O     "Blend_T-20".Dose.Dose_Header_Req.%X24;  //Header 2 Req
      =     "Blend to Preparation"."T-20".Raw_Material.HW.Header2_Req;

      L     "Blend to Preparation".Recipe."T-20".HW.Sp_Flush_to_BlendQty;  //Load Flush to Blend Sp Dose From Recipe
      T     "Blend_T-20"."HW Flushing".Qty."Flush to Blend Qty";
      L     "Blend to Preparation".Recipe."T-20".HW.Sp_Flush_to_DrainQty;  //Load Flush to Blend Sp Dose From Recipe
      T     "Blend_T-20"."HW Flushing".Qty."Flush to Drain Qty";  //Load Drain Time from recipe
      L     "Blend to Preparation".Recipe."T-20".HW.Sp_DrainTime;
      T     "Blend_T-20"."HW Flushing".TimeDrain_SP;

      L     "Blend_T-20".Dose_HW.P_SPEED;  //Pump Speed
      T     "Blend to Preparation".Recipe."T-20".HW.SP_PumpSpeed;

//General
      O     "Blend_T-20".IN_FBAV_Header1;
      =     "Blend to Preparation"."T-20".LineHeader1_OK;
      O     "Blend_T-20".IN_FBAV_Header2;
      =     "Blend to Preparation"."T-20".LineHeader2_OK;
      O     "Blend_T-20".IN_FBAV_Vinegar;
      =     "Blend to Preparation"."T-20".LineVinegar_OK;


NETWORK
TITLE = ChiliAwetan1 to Blending T-21
//Valve Open
      A     "Preparation to Blend"."T-02_ChiliAwetan_1".Valve_Open;
      A(;
      O(;
      A     "Blend_T-21".Dose.Dose_Header_Req.%X0;
      A     "Blend_T-21".IN_FBAV_Header1;
      );
      O(;
      A     "Blend_T-21".Dose.Dose_Header_Req.%X16;
      A     "Blend_T-21".IN_FBAV_Header2;
      );
      );
      =     "Blend_T-21".Dose_ChiliAwetan1.V_OPEN;
//Pump On
      O     "Preparation to Blend"."T-02_ChiliAwetan_1".Pump_Run;
      =     "Blend_T-21".Dose_ChiliAwetan1.P_RUN;
//Tank Available
      O     "Preparation to Blend"."T-02_ChiliAwetan_1".Tank_Available;
      O     "Blend_T-21".Dose_ChiliAwetan1.QDOSERun;
      =     "Blend_T-21".Dose.Dose_Tank_Available.%X0;
//Product Ready
      O     "Preparation to Blend"."T-02_ChiliAwetan_1".Product_Ready;
      =     "Blend_T-21".Dose.Dose_Prod_Ready.%X0;
//Level Tank
      L     "Preparation to Blend"."T-02_ChiliAwetan_1".Level;
      T     "Blend_T-21"."Dose_Level_%"."ChiliAwetan1%";


NETWORK
TITLE = ChiliAwetan2 to Blending T-21
//Valve Open
      A     "Preparation to Blend"."T-03_ChiliAwetan_2".Valve_Open;
      A(;
      O(;
      A     "Blend_T-21".Dose.Dose_Header_Req.%X1;
      A     "Blend_T-21".IN_FBAV_Header1;
      );
      O(;
      A     "Blend_T-21".Dose.Dose_Header_Req.%X17;
      A     "Blend_T-21".IN_FBAV_Header2;
      );
      );
      =     "Blend_T-21".Dose_ChiliAwetan2.V_OPEN;
//Pump On
      O     "Preparation to Blend"."T-03_ChiliAwetan_2".Pump_Run;
      =     "Blend_T-21".Dose_ChiliAwetan2.P_RUN;
//Tank Available
      O     "Preparation to Blend"."T-03_ChiliAwetan_2".Tank_Available;
      O     "Blend_T-21".Dose_ChiliAwetan2.QDOSERun;
      =     "Blend_T-21".Dose.Dose_Tank_Available.%X1;
//Product Ready
      O     "Preparation to Blend"."T-03_ChiliAwetan_2".Product_Ready;
      =     "Blend_T-21".Dose.Dose_Prod_Ready.%X1;
//Level Tank
      L     "Preparation to Blend"."T-03_ChiliAwetan_2".Level;
      T     "Blend_T-21"."Dose_Level_%"."ChiliAwetan2%";


NETWORK
TITLE = ChiliAwetan3 to Blending T-21
//Valve Open
      A     "Preparation to Blend"."T-04_ChiliAwetan_3".Valve_Open;
      A(;
      O(;
      A     "Blend_T-21".Dose.Dose_Header_Req.%X2;
      A     "Blend_T-21".IN_FBAV_Header1;
      );
      O(;
      A     "Blend_T-21".Dose.Dose_Header_Req.%X18;
      A     "Blend_T-21".IN_FBAV_Header2;
      );
      );
      =     "Blend_T-21".Dose_ChiliAwetan3.V_OPEN;
//Pump On
      O     "Preparation to Blend"."T-04_ChiliAwetan_3".Pump_Run;
      =     "Blend_T-21".Dose_ChiliAwetan3.P_RUN;
//Tank Available
      O     "Preparation to Blend"."T-04_ChiliAwetan_3".Tank_Available;
      O     "Blend_T-21".Dose_ChiliAwetan3.QDOSERun;
      =     "Blend_T-21".Dose.Dose_Tank_Available.%X2;
//Product Ready
      O     "Preparation to Blend"."T-04_ChiliAwetan_3".Product_Ready;
      =     "Blend_T-21".Dose.Dose_Prod_Ready.%X2;
//Level Tank
      L     "Preparation to Blend"."T-04_ChiliAwetan_3".Level;
      T     "Blend_T-21"."Dose_Level_%"."ChiliAwetan3%";


NETWORK
TITLE = Tomato to Blending T-21
//Valve Open
      A     "Preparation to Blend"."T-05_Tomato".Valve_Open;
      A(;
      O(;
      A     "Blend_T-21".Dose.Dose_Header_Req.%X3;
      A     "Blend_T-21".IN_FBAV_Header1;
      );
      O(;
      A     "Blend_T-21".Dose.Dose_Header_Req.%X19;
      A     "Blend_T-21".IN_FBAV_Header2;
      );
      );
      =     "Blend_T-21".Dose_Tomato.V_OPEN;
//Pump On
      O     "Preparation to Blend"."T-05_Tomato".Pump_Run;
      =     "Blend_T-21".Dose_Tomato.P_RUN;
//Tank Available
      O     "Preparation to Blend"."T-05_Tomato".Tank_Available;
      O     "Blend_T-21".Dose_Tomato.QDOSERun;
      =     "Blend_T-21".Dose.Dose_Tank_Available.%X3;
//Product Ready
      O     "Preparation to Blend"."T-05_Tomato".Product_Ready;
      =     "Blend_T-21".Dose.Dose_Prod_Ready.%X3;
//Level Tank
      L     "Preparation to Blend"."T-05_Tomato".Level;
      T     "Blend_T-21"."Dose_Level_%"."Tomato%";


NETWORK
TITLE = ChiliFresh1 to Blending T-21
//Valve Open
      A     "Preparation to Blend"."T-06_ChiliFresh_1".Valve_Open;
      A(;
      O(;
      A     "Blend_T-21".Dose.Dose_Header_Req.%X4;
      A     "Blend_T-21".IN_FBAV_Header1;
      );
      O(;
      A     "Blend_T-21".Dose.Dose_Header_Req.%X20;
      A     "Blend_T-21".IN_FBAV_Header2;
      );
      );
      =     "Blend_T-21".Dose_ChiliFresh1.V_OPEN;
//Pump On
      O     "Preparation to Blend"."T-06_ChiliFresh_1".Pump_Run;
      =     "Blend_T-21".Dose_ChiliFresh1.P_RUN;
//Tank Available
      O     "Preparation to Blend"."T-06_ChiliFresh_1".Tank_Available;
      O     "Blend_T-21".Dose_ChiliFresh1.QDOSERun;
      =     "Blend_T-21".Dose.Dose_Tank_Available.%X4;
//Product Ready
      O     "Preparation to Blend"."T-06_ChiliFresh_1".Product_Ready;
      =     "Blend_T-21".Dose.Dose_Prod_Ready.%X4;
//Level Tank
      L     "Preparation to Blend"."T-06_ChiliFresh_1".Level;
      T     "Blend_T-21"."Dose_Level_%"."ChiliFresh1%";


NETWORK
TITLE = ChiliFresh2 to Blending T-21
//Valve Open
      A     "Preparation to Blend"."T-07_ChiliFresh_2".Valve_Open;
      A(;
      O(;
      A     "Blend_T-21".Dose.Dose_Header_Req.%X5;
      A     "Blend_T-21".IN_FBAV_Header1;
      );
      O(;
      A     "Blend_T-21".Dose.Dose_Header_Req.%X21;
      A     "Blend_T-21".IN_FBAV_Header2;
      );
      );
      =     "Blend_T-21".Dose_ChiliFresh2.V_OPEN;
//Pump On
      O     "Preparation to Blend"."T-07_ChiliFresh_2".Pump_Run;
      =     "Blend_T-21".Dose_ChiliFresh2.P_RUN;
//Tank Available
      O     "Preparation to Blend"."T-07_ChiliFresh_2".Tank_Available;
      O     "Blend_T-21".Dose_ChiliFresh2.QDOSERun;
      =     "Blend_T-21".Dose.Dose_Tank_Available.%X5;
//Product Ready
      O     "Preparation to Blend"."T-07_ChiliFresh_2".Product_Ready;
      =     "Blend_T-21".Dose.Dose_Prod_Ready.%X5;
//Level Tank
      L     "Preparation to Blend"."T-07_ChiliFresh_2".Level;
      T     "Blend_T-21"."Dose_Level_%"."ChiliFresh2%";


NETWORK
TITLE = ChiliFresh3 to Blending T-21
//Valve Open
      A     "Preparation to Blend"."T-08_ChiliFresh_3".Valve_Open;
      A(;
      O(;
      A     "Blend_T-21".Dose.Dose_Header_Req.%X6;
      A     "Blend_T-21".IN_FBAV_Header1;
      );
      O(;
      A     "Blend_T-21".Dose.Dose_Header_Req.%X22;
      A     "Blend_T-21".IN_FBAV_Header2;
      );
      );
      =     "Blend_T-21".Dose_ChiliFresh3.V_OPEN;
//Pump On
      O     "Preparation to Blend"."T-08_ChiliFresh_3".Pump_Run;
      =     "Blend_T-21".Dose_ChiliFresh3.P_RUN;
//Tank Available
      O     "Preparation to Blend"."T-08_ChiliFresh_3".Tank_Available;
      O     "Blend_T-21".Dose_ChiliFresh3.QDOSERun;
      =     "Blend_T-21".Dose.Dose_Tank_Available.%X6;
//Product Ready
      O     "Preparation to Blend"."T-08_ChiliFresh_3".Product_Ready;
      =     "Blend_T-21".Dose.Dose_Prod_Ready.%X6;
//Level Tank
      L     "Preparation to Blend"."T-08_ChiliFresh_3".Level;
      T     "Blend_T-21"."Dose_Level_%"."ChiliFresh3%";


NETWORK
TITLE = Garlic to Blending T-21
//Valve Open
      A     "Preparation to Blend"."T-09_Garlic".Valve_Open;
      A(;
      O(;
      A     "Blend_T-21".Dose.Dose_Header_Req.%X7;
      A     "Blend_T-21".IN_FBAV_Header1;
      );
      O(;
      A     "Blend_T-21".Dose.Dose_Header_Req.%X23;
      A     "Blend_T-21".IN_FBAV_Header2;
      );
      );
      =     "Blend_T-21".Dose_Garlic.V_OPEN;
//Pump On
      O     "Preparation to Blend"."T-09_Garlic".Pump_Run;
      =     "Blend_T-21".Dose_Garlic.P_RUN;
//Tank Available
      O     "Preparation to Blend"."T-09_Garlic".Tank_Available;
      O     "Blend_T-21".Dose_Garlic.QDOSERun;
      =     "Blend_T-21".Dose.Dose_Tank_Available.%X7;
//Product Ready
      O     "Preparation to Blend"."T-09_Garlic".Product_Ready;
      =     "Blend_T-21".Dose.Dose_Prod_Ready.%X7;
//Level Tank
      L     "Preparation to Blend"."T-09_Garlic".Level;
      T     "Blend_T-21"."Dose_Level_%"."Garlic%";


NETWORK
TITLE = Vinegar to Blending T-21
//Valve Open
      A     "Preparation to Blend"."T-10_Vinegar".Valve_Open;
      A     "Blend_T-21".IN_FBAV_Vinegar;
      =     "Blend_T-21".Dose_Vinegar.V_OPEN;
//Pump On
      O     "Preparation to Blend"."T-10_Vinegar".Pump_Run;
      =     "Blend_T-21".Dose_Vinegar.P_RUN;
//Tank Available
      O     "Preparation to Blend"."T-10_Vinegar".Tank_Available;
      O     "Blend_T-21".Dose_Vinegar.QDOSERun;
      =     "Blend_T-21".Dose.Dose_Tank_Available.%X9;
//Product Ready
      O     "Preparation to Blend"."T-10_Vinegar".Product_Ready;
      =     "Blend_T-21".Dose.Dose_Prod_Ready.%X9;
//Level Tank
      L     "Preparation to Blend"."T-10_Vinegar".Level;
      T     "Blend_T-21"."Dose_Level_%"."Vinegar%";


